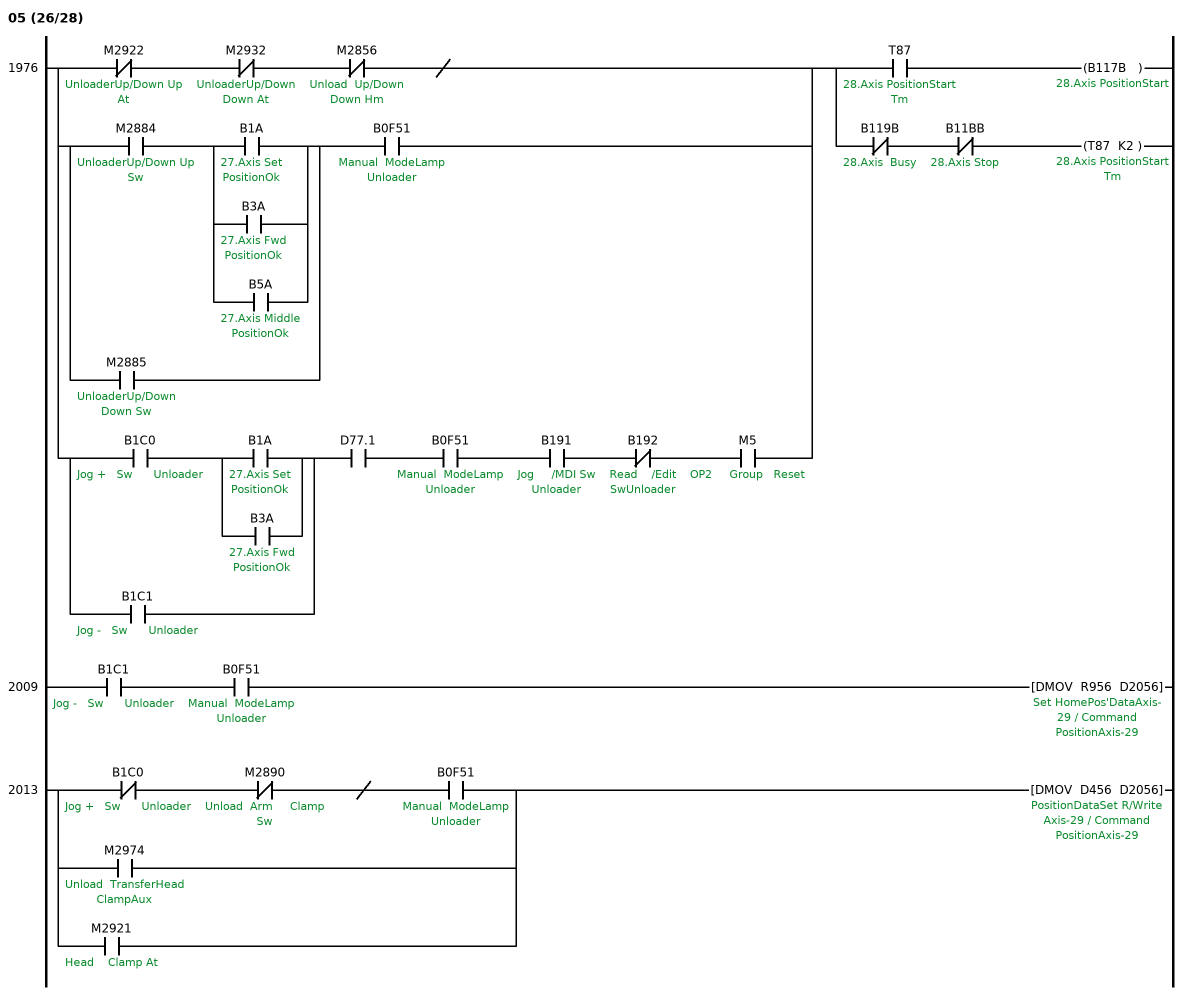
1976  LDI     M2922  ; UnloaderUp/Down Up At
      ANI     M2932  ; UnloaderUp/Down Down At
      ANI     M2856  ; Unload  Up/Down Down Hm
      INV
      LD      M2884  ; UnloaderUp/Down Up Sw
      LD      B1A  ; 27.Axis Set     PositionOk
      OR      B3A  ; 27.Axis Fwd     PositionOk
      OR      B5A  ; 27.Axis Middle  PositionOk
      ANB
      OR      M2885  ; UnloaderUp/Down Down Sw
      AND     B0F51  ; Manual  ModeLampUnloader
      ORB
      LD      B1C0  ; Jog +   Sw      Unloader
      LD      B1A  ; 27.Axis Set     PositionOk
      OR      B3A  ; 27.Axis Fwd     PositionOk
      ANB
      OR      B1C1  ; Jog -   Sw      Unloader
      AND     D77.1
      AND     B0F51  ; Manual  ModeLampUnloader
      AND     B191  ; Jog     /MDI Sw Unloader
      ANI     B192  ; Read    /Edit SwUnloader
      AND     M5  ; OP2     Group   Reset
      ORB
      MPS
      AND     T87  ; 28.Axis PositionStart Tm
      OUT     B117B  ; 28.Axis PositionStart
      MPP
      ANI     B119B  ; 28.Axis  Busy
      ANI     B11BB  ; 28.Axis Stop
      OUT     T87 K2  ; 28.Axis PositionStart Tm
2009  LD      B1C1  ; Jog -   Sw      Unloader
      AND     B0F51  ; Manual  ModeLampUnloader
      DMOV    R956 D2056  ; Set HomePos'DataAxis-29 / Command PositionAxis-29
2013  LDI     B1C0  ; Jog +   Sw      Unloader
      ANI     M2890  ; Unload  Arm     Clamp Sw
      INV
      AND     B0F51  ; Manual  ModeLampUnloader
      OR      M2974  ; Unload  TransferHead    ClampAux
      OR      M2921  ; Head    Clamp At
      DMOV    D456 D2056  ; PositionDataSet R/Write Axis-29
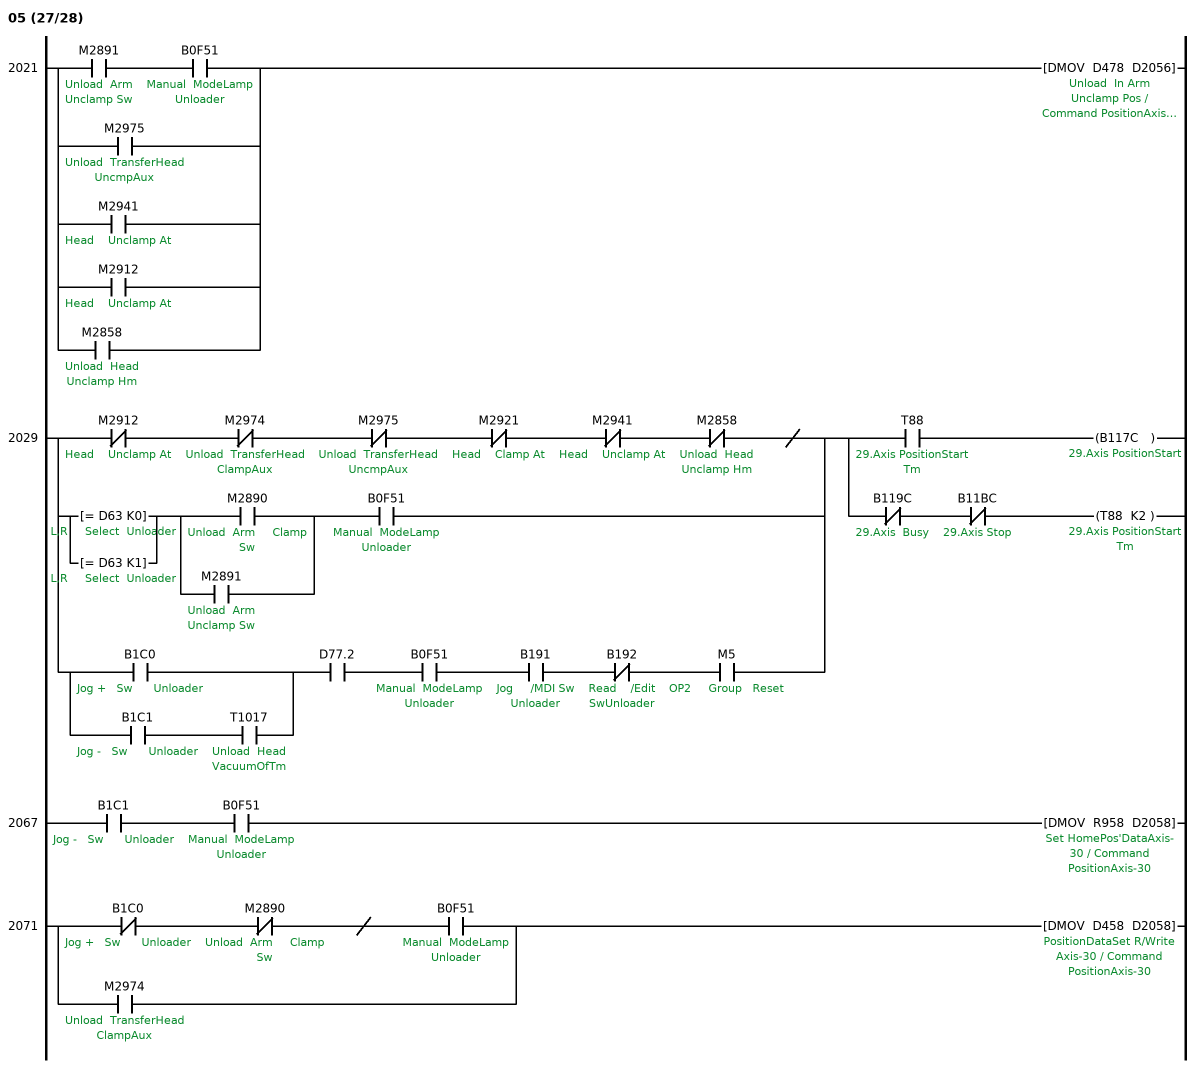
2021  LD      M2891  ; Unload  Arm     Unclamp Sw
      AND     B0F51  ; Manual  ModeLampUnloader
      OR      M2975  ; Unload  TransferHead    UncmpAux
      OR      M2941  ; Head    Unclamp At
      OR      M2912  ; Head    Unclamp At
      OR      M2858  ; Unload  Head    Unclamp Hm
      DMOV    D478 D2056  ; Unload  In Arm  Unclamp Pos
2029  LDI     M2912  ; Head    Unclamp At
      ANI     M2974  ; Unload  TransferHead    ClampAux
      ANI     M2975  ; Unload  TransferHead    UncmpAux
      ANI     M2921  ; Head    Clamp At
      ANI     M2941  ; Head    Unclamp At
      ANI     M2858  ; Unload  Head    Unclamp Hm
      INV
      LD=     D63 K0  ; L,R     Select  Unloader
      OR=     D63 K1  ; L,R     Select  Unloader
      LD      M2890  ; Unload  Arm     Clamp Sw
      OR      M2891  ; Unload  Arm     Unclamp Sw
      ANB
      AND     B0F51  ; Manual  ModeLampUnloader
      ORB
      LD      B1C0  ; Jog +   Sw      Unloader
      LD      B1C1  ; Jog -   Sw      Unloader
      AND     T1017  ; Unload  Head    VacuumOfTm
      ORB
      AND     D77.2
      AND     B0F51  ; Manual  ModeLampUnloader
      AND     B191  ; Jog     /MDI Sw Unloader
      ANI     B192  ; Read    /Edit SwUnloader
      AND     M5  ; OP2     Group   Reset
      ORB
      MPS
      AND     T88  ; 29.Axis PositionStart Tm
      OUT     B117C  ; 29.Axis PositionStart
      MPP
      ANI     B119C  ; 29.Axis  Busy
      ANI     B11BC  ; 29.Axis Stop
      OUT     T88 K2  ; 29.Axis PositionStart Tm
2067  LD      B1C1  ; Jog -   Sw      Unloader
      AND     B0F51  ; Manual  ModeLampUnloader
      DMOV    R958 D2058  ; Set HomePos'DataAxis-30 / Command PositionAxis-30
2071  LDI     B1C0  ; Jog +   Sw      Unloader
      ANI     M2890  ; Unload  Arm     Clamp Sw
      INV
      AND     B0F51  ; Manual  ModeLampUnloader
      OR      M2974  ; Unload  TransferHead    ClampAux
      DMOV    D458 D2058  ; PositionDataSet R/Write Axis-30
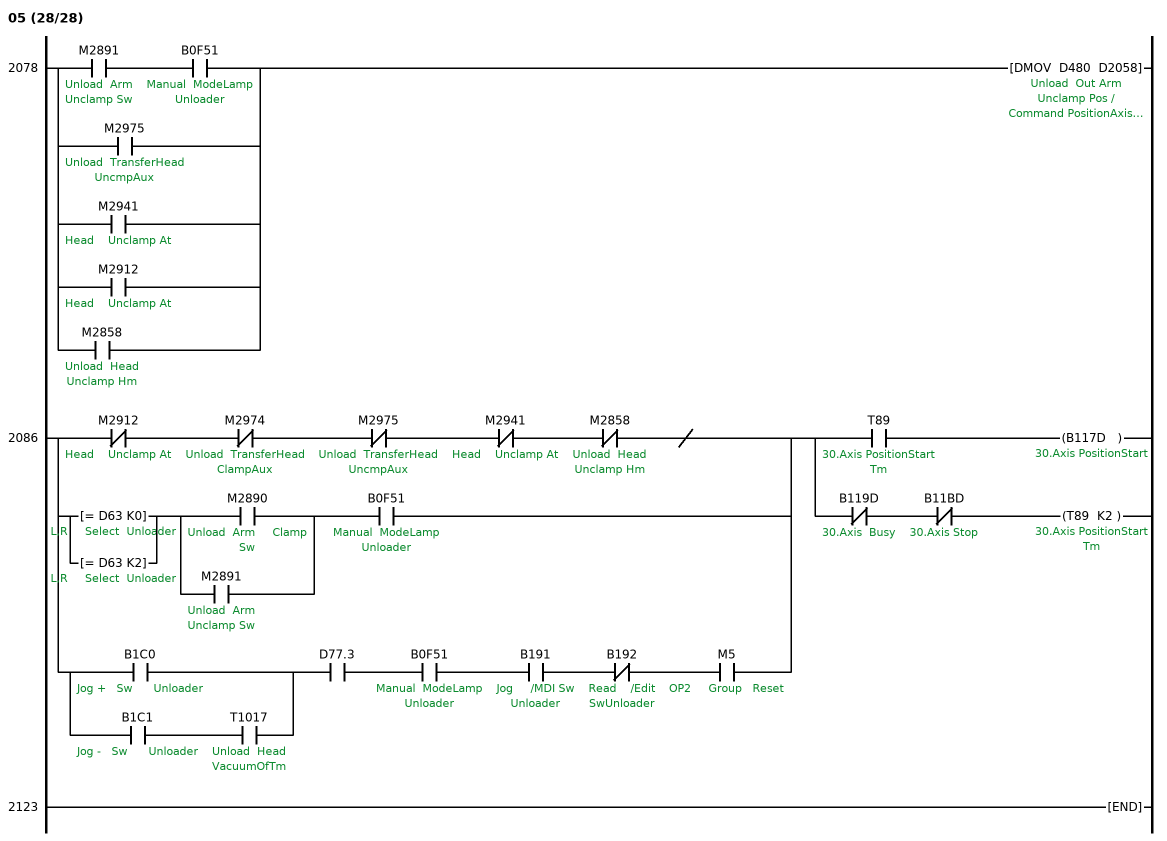
2078  LD      M2891  ; Unload  Arm     Unclamp Sw
      AND     B0F51  ; Manual  ModeLampUnloader
      OR      M2975  ; Unload  TransferHead    UncmpAux
      OR      M2941  ; Head    Unclamp At
      OR      M2912  ; Head    Unclamp At
      OR      M2858  ; Unload  Head    Unclamp Hm
      DMOV    D480 D2058  ; Unload  Out Arm Unclamp Pos
2086  LDI     M2912  ; Head    Unclamp At
      ANI     M2974  ; Unload  TransferHead    ClampAux
      ANI     M2975  ; Unload  TransferHead    UncmpAux
      ANI     M2941  ; Head    Unclamp At
      ANI     M2858  ; Unload  Head    Unclamp Hm
      INV
      LD=     D63 K0  ; L,R     Select  Unloader
      OR=     D63 K2  ; L,R     Select  Unloader
      LD      M2890  ; Unload  Arm     Clamp Sw
      OR      M2891  ; Unload  Arm     Unclamp Sw
      ANB
      AND     B0F51  ; Manual  ModeLampUnloader
      ORB
      LD      B1C0  ; Jog +   Sw      Unloader
      LD      B1C1  ; Jog -   Sw      Unloader
      AND     T1017  ; Unload  Head    VacuumOfTm
      ORB
      AND     D77.3
      AND     B0F51  ; Manual  ModeLampUnloader
      AND     B191  ; Jog     /MDI Sw Unloader
      ANI     B192  ; Read    /Edit SwUnloader
      AND     M5  ; OP2     Group   Reset
      ORB
      MPS
      AND     T89  ; 30.Axis PositionStart Tm
      OUT     B117D  ; 30.Axis PositionStart
      MPP
      ANI     B119D  ; 30.Axis  Busy
      ANI     B11BD  ; 30.Axis Stop
      OUT     T89 K2  ; 30.Axis PositionStart Tm
2123  END
END_PROGRAM

PROGRAM 06  // Servo Part
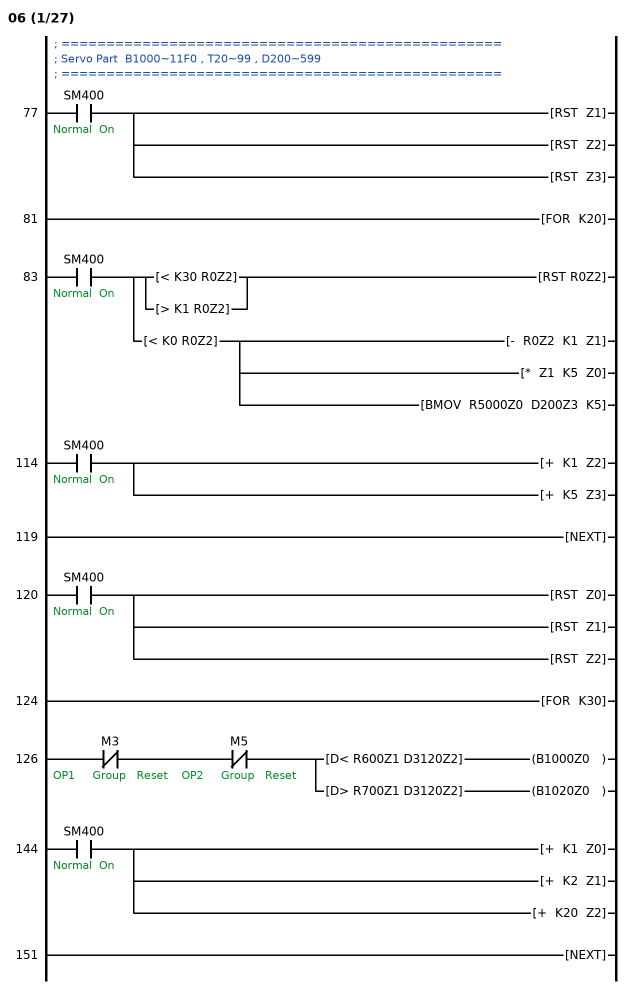
; =================================================
; Servo Part  B1000~11F0 , T20~99 , D200~599
; =================================================
77    LD      SM400  ; Normal  On
      RST     Z1
      RST     Z2
      RST     Z3
81    FOR     K20
83    LD      SM400  ; Normal  On
      MPS
      LD<     K30 R0Z2
      OR>     K1 R0Z2
      ANB
      RST     R0Z2
      MPP
      AND<    K0 R0Z2
      -       R0Z2 K1 Z1
      *       Z1 K5 Z0
      BMOV    R5000Z0 D200Z3 K5
114   LD      SM400  ; Normal  On
      +       K1 Z2
      +       K5 Z3
119   NEXT
120   LD      SM400  ; Normal  On
      RST     Z0
      RST     Z1
      RST     Z2
124   FOR     K30
126   LDI     M3  ; OP1     Group   Reset
      ANI     M5  ; OP2     Group   Reset
      MPS
      ANDD<   R600Z1 D3120Z2
      OUT     B1000Z0
      MPP
      ANDD>   R700Z1 D3120Z2
      OUT     B1020Z0
144   LD      SM400  ; Normal  On
      +       K1 Z0
      +       K2 Z1
      +       K20 Z2
151   NEXT
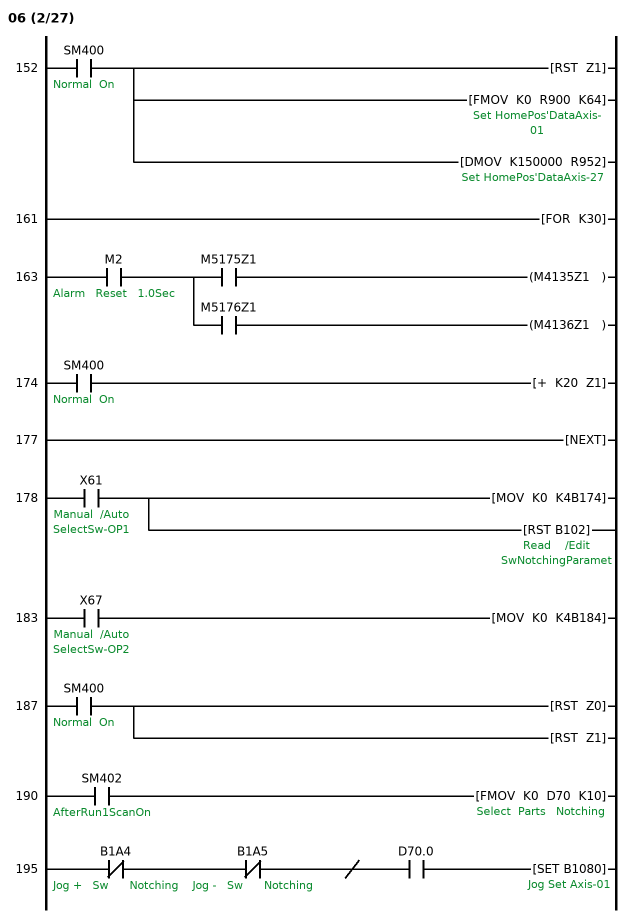
152   LD      SM400  ; Normal  On
      RST     Z1
      FMOV    K0 R900 K64  ; Set HomePos'DataAxis-01
      DMOV    K150000 R952  ; Set HomePos'DataAxis-27
161   FOR     K30
163   LD      M2  ; Alarm   Reset   1.0Sec
      MPS
      AND     M5175Z1
      OUT     M4135Z1
      MPP
      AND     M5176Z1
      OUT     M4136Z1
174   LD      SM400  ; Normal  On
      +       K20 Z1
177   NEXT
178   LD      X61  ; Manual  /Auto   SelectSw-OP1
      MOV     K0 K4B174  ; Jog FastSpeed SwNotching
      RST     B102  ; Read    /Edit SwNotchingParamet
183   LD      X67  ; Manual  /Auto   SelectSw-OP2
      MOV     K0 K4B184  ; Jog FastSpeed SwL & Z
187   LD      SM400  ; Normal  On
      RST     Z0
      RST     Z1
190   LD      SM402  ; AfterRun1ScanOn
      FMOV    K0 D70 K10  ; Select  Parts   Notching
195   LDI     B1A4  ; Jog +   Sw      Notching
      ANI     B1A5  ; Jog -   Sw      Notching
      INV
      AND     D70.0
      SET     B1080  ; Jog Set Axis-01
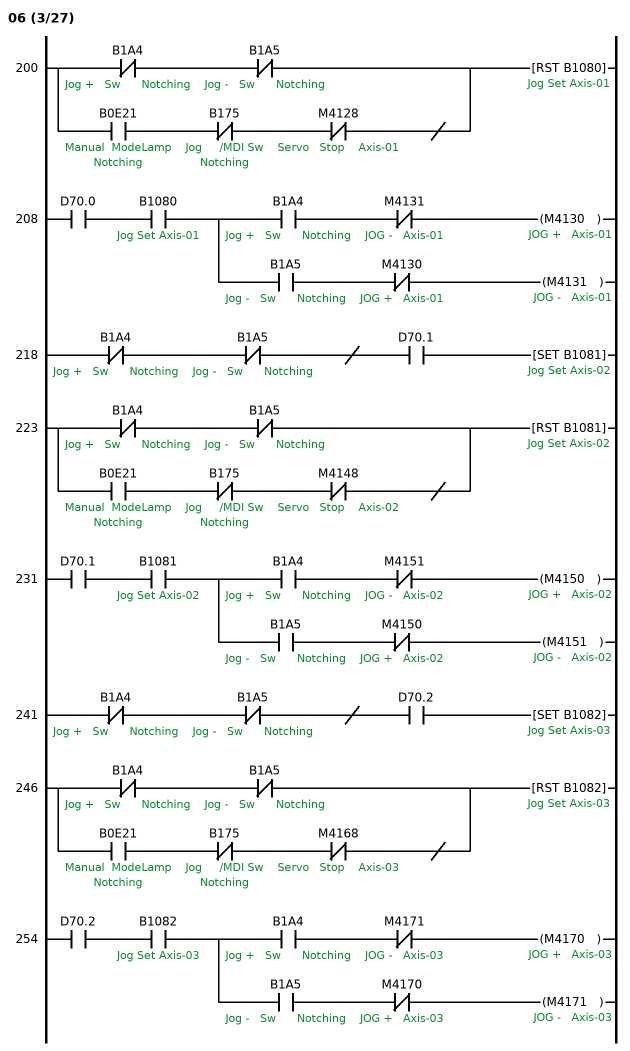
200   LDI     B1A4  ; Jog +   Sw      Notching
      ANI     B1A5  ; Jog -   Sw      Notching
      LD      B0E21  ; Manual  ModeLampNotching
      ANI     B175  ; Jog     /MDI Sw Notching
      ANI     M4128  ; Servo   Stop    Axis-01
      INV
      ORB
      RST     B1080  ; Jog Set Axis-01
208   LD      D70.0
      AND     B1080  ; Jog Set Axis-01
      MPS
      AND     B1A4  ; Jog +   Sw      Notching
      ANI     M4131  ; JOG -   Axis-01
      OUT     M4130  ; JOG +   Axis-01
      MPP
      AND     B1A5  ; Jog -   Sw      Notching
      ANI     M4130  ; JOG +   Axis-01
      OUT     M4131  ; JOG -   Axis-01
218   LDI     B1A4  ; Jog +   Sw      Notching
      ANI     B1A5  ; Jog -   Sw      Notching
      INV
      AND     D70.1
      SET     B1081  ; Jog Set Axis-02
223   LDI     B1A4  ; Jog +   Sw      Notching
      ANI     B1A5  ; Jog -   Sw      Notching
      LD      B0E21  ; Manual  ModeLampNotching
      ANI     B175  ; Jog     /MDI Sw Notching
      ANI     M4148  ; Servo   Stop    Axis-02
      INV
      ORB
      RST     B1081  ; Jog Set Axis-02
231   LD      D70.1
      AND     B1081  ; Jog Set Axis-02
      MPS
      AND     B1A4  ; Jog +   Sw      Notching
      ANI     M4151  ; JOG -   Axis-02
      OUT     M4150  ; JOG +   Axis-02
      MPP
      AND     B1A5  ; Jog -   Sw      Notching
      ANI     M4150  ; JOG +   Axis-02
      OUT     M4151  ; JOG -   Axis-02
241   LDI     B1A4  ; Jog +   Sw      Notching
      ANI     B1A5  ; Jog -   Sw      Notching
      INV
      AND     D70.2
      SET     B1082  ; Jog Set Axis-03
246   LDI     B1A4  ; Jog +   Sw      Notching
      ANI     B1A5  ; Jog -   Sw      Notching
      LD      B0E21  ; Manual  ModeLampNotching
      ANI     B175  ; Jog     /MDI Sw Notching
      ANI     M4168  ; Servo   Stop    Axis-03
      INV
      ORB
      RST     B1082  ; Jog Set Axis-03
254   LD      D70.2
      AND     B1082  ; Jog Set Axis-03
      MPS
      AND     B1A4  ; Jog +   Sw      Notching
      ANI     M4171  ; JOG -   Axis-03
      OUT     M4170  ; JOG +   Axis-03
      MPP
      AND     B1A5  ; Jog -   Sw      Notching
      ANI     M4170  ; JOG +   Axis-03
      OUT     M4171  ; JOG -   Axis-03
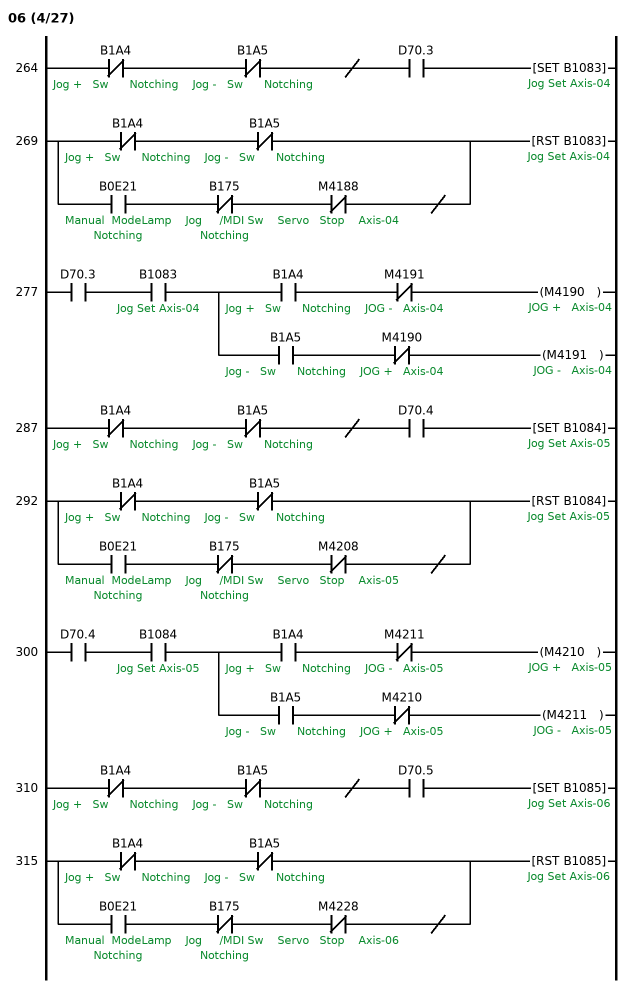
264   LDI     B1A4  ; Jog +   Sw      Notching
      ANI     B1A5  ; Jog -   Sw      Notching
      INV
      AND     D70.3
      SET     B1083  ; Jog Set Axis-04
269   LDI     B1A4  ; Jog +   Sw      Notching
      ANI     B1A5  ; Jog -   Sw      Notching
      LD      B0E21  ; Manual  ModeLampNotching
      ANI     B175  ; Jog     /MDI Sw Notching
      ANI     M4188  ; Servo   Stop    Axis-04
      INV
      ORB
      RST     B1083  ; Jog Set Axis-04
277   LD      D70.3
      AND     B1083  ; Jog Set Axis-04
      MPS
      AND     B1A4  ; Jog +   Sw      Notching
      ANI     M4191  ; JOG -   Axis-04
      OUT     M4190  ; JOG +   Axis-04
      MPP
      AND     B1A5  ; Jog -   Sw      Notching
      ANI     M4190  ; JOG +   Axis-04
      OUT     M4191  ; JOG -   Axis-04
287   LDI     B1A4  ; Jog +   Sw      Notching
      ANI     B1A5  ; Jog -   Sw      Notching
      INV
      AND     D70.4
      SET     B1084  ; Jog Set Axis-05
292   LDI     B1A4  ; Jog +   Sw      Notching
      ANI     B1A5  ; Jog -   Sw      Notching
      LD      B0E21  ; Manual  ModeLampNotching
      ANI     B175  ; Jog     /MDI Sw Notching
      ANI     M4208  ; Servo   Stop    Axis-05
      INV
      ORB
      RST     B1084  ; Jog Set Axis-05
300   LD      D70.4
      AND     B1084  ; Jog Set Axis-05
      MPS
      AND     B1A4  ; Jog +   Sw      Notching
      ANI     M4211  ; JOG -   Axis-05
      OUT     M4210  ; JOG +   Axis-05
      MPP
      AND     B1A5  ; Jog -   Sw      Notching
      ANI     M4210  ; JOG +   Axis-05
      OUT     M4211  ; JOG -   Axis-05
310   LDI     B1A4  ; Jog +   Sw      Notching
      ANI     B1A5  ; Jog -   Sw      Notching
      INV
      AND     D70.5
      SET     B1085  ; Jog Set Axis-06
315   LDI     B1A4  ; Jog +   Sw      Notching
      ANI     B1A5  ; Jog -   Sw      Notching
      LD      B0E21  ; Manual  ModeLampNotching
      ANI     B175  ; Jog     /MDI Sw Notching
      ANI     M4228  ; Servo   Stop    Axis-06
      INV
      ORB
      RST     B1085  ; Jog Set Axis-06
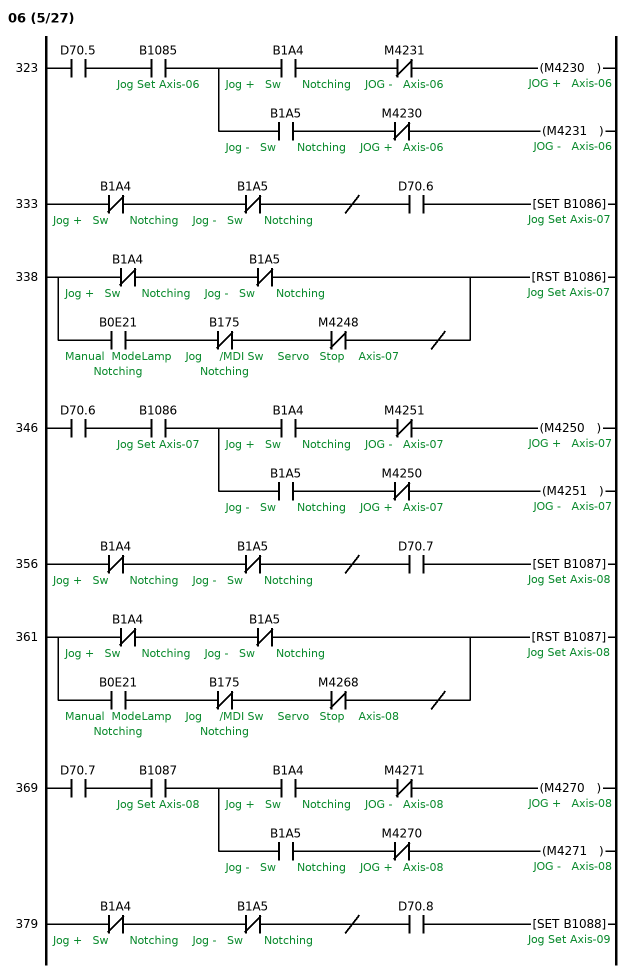
323   LD      D70.5
      AND     B1085  ; Jog Set Axis-06
      MPS
      AND     B1A4  ; Jog +   Sw      Notching
      ANI     M4231  ; JOG -   Axis-06
      OUT     M4230  ; JOG +   Axis-06
      MPP
      AND     B1A5  ; Jog -   Sw      Notching
      ANI     M4230  ; JOG +   Axis-06
      OUT     M4231  ; JOG -   Axis-06
333   LDI     B1A4  ; Jog +   Sw      Notching
      ANI     B1A5  ; Jog -   Sw      Notching
      INV
      AND     D70.6
      SET     B1086  ; Jog Set Axis-07
338   LDI     B1A4  ; Jog +   Sw      Notching
      ANI     B1A5  ; Jog -   Sw      Notching
      LD      B0E21  ; Manual  ModeLampNotching
      ANI     B175  ; Jog     /MDI Sw Notching
      ANI     M4248  ; Servo   Stop    Axis-07
      INV
      ORB
      RST     B1086  ; Jog Set Axis-07
346   LD      D70.6
      AND     B1086  ; Jog Set Axis-07
      MPS
      AND     B1A4  ; Jog +   Sw      Notching
      ANI     M4251  ; JOG -   Axis-07
      OUT     M4250  ; JOG +   Axis-07
      MPP
      AND     B1A5  ; Jog -   Sw      Notching
      ANI     M4250  ; JOG +   Axis-07
      OUT     M4251  ; JOG -   Axis-07
356   LDI     B1A4  ; Jog +   Sw      Notching
      ANI     B1A5  ; Jog -   Sw      Notching
      INV
      AND     D70.7
      SET     B1087  ; Jog Set Axis-08
361   LDI     B1A4  ; Jog +   Sw      Notching
      ANI     B1A5  ; Jog -   Sw      Notching
      LD      B0E21  ; Manual  ModeLampNotching
      ANI     B175  ; Jog     /MDI Sw Notching
      ANI     M4268  ; Servo   Stop    Axis-08
      INV
      ORB
      RST     B1087  ; Jog Set Axis-08
369   LD      D70.7
      AND     B1087  ; Jog Set Axis-08
      MPS
      AND     B1A4  ; Jog +   Sw      Notching
      ANI     M4271  ; JOG -   Axis-08
      OUT     M4270  ; JOG +   Axis-08
      MPP
      AND     B1A5  ; Jog -   Sw      Notching
      ANI     M4270  ; JOG +   Axis-08
      OUT     M4271  ; JOG -   Axis-08
379   LDI     B1A4  ; Jog +   Sw      Notching
      ANI     B1A5  ; Jog -   Sw      Notching
      INV
      AND     D70.8
      SET     B1088  ; Jog Set Axis-09
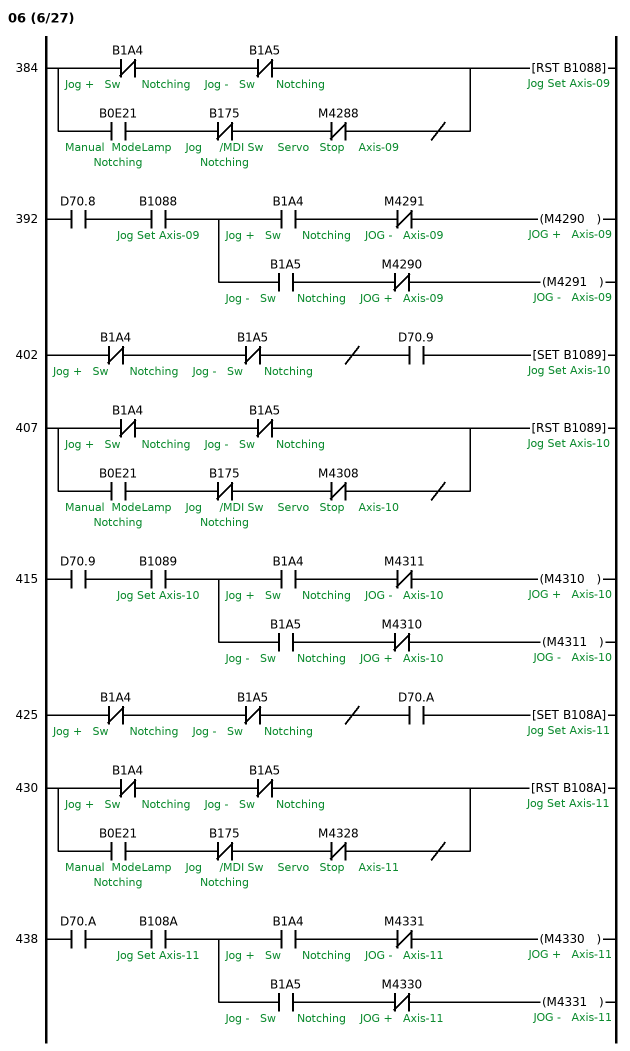
384   LDI     B1A4  ; Jog +   Sw      Notching
      ANI     B1A5  ; Jog -   Sw      Notching
      LD      B0E21  ; Manual  ModeLampNotching
      ANI     B175  ; Jog     /MDI Sw Notching
      ANI     M4288  ; Servo   Stop    Axis-09
      INV
      ORB
      RST     B1088  ; Jog Set Axis-09
392   LD      D70.8
      AND     B1088  ; Jog Set Axis-09
      MPS
      AND     B1A4  ; Jog +   Sw      Notching
      ANI     M4291  ; JOG -   Axis-09
      OUT     M4290  ; JOG +   Axis-09
      MPP
      AND     B1A5  ; Jog -   Sw      Notching
      ANI     M4290  ; JOG +   Axis-09
      OUT     M4291  ; JOG -   Axis-09
402   LDI     B1A4  ; Jog +   Sw      Notching
      ANI     B1A5  ; Jog -   Sw      Notching
      INV
      AND     D70.9
      SET     B1089  ; Jog Set Axis-10
407   LDI     B1A4  ; Jog +   Sw      Notching
      ANI     B1A5  ; Jog -   Sw      Notching
      LD      B0E21  ; Manual  ModeLampNotching
      ANI     B175  ; Jog     /MDI Sw Notching
      ANI     M4308  ; Servo   Stop    Axis-10
      INV
      ORB
      RST     B1089  ; Jog Set Axis-10
415   LD      D70.9
      AND     B1089  ; Jog Set Axis-10
      MPS
      AND     B1A4  ; Jog +   Sw      Notching
      ANI     M4311  ; JOG -   Axis-10
      OUT     M4310  ; JOG +   Axis-10
      MPP
      AND     B1A5  ; Jog -   Sw      Notching
      ANI     M4310  ; JOG +   Axis-10
      OUT     M4311  ; JOG -   Axis-10
425   LDI     B1A4  ; Jog +   Sw      Notching
      ANI     B1A5  ; Jog -   Sw      Notching
      INV
      AND     D70.A
      SET     B108A  ; Jog Set Axis-11
430   LDI     B1A4  ; Jog +   Sw      Notching
      ANI     B1A5  ; Jog -   Sw      Notching
      LD      B0E21  ; Manual  ModeLampNotching
      ANI     B175  ; Jog     /MDI Sw Notching
      ANI     M4328  ; Servo   Stop    Axis-11
      INV
      ORB
      RST     B108A  ; Jog Set Axis-11
438   LD      D70.A
      AND     B108A  ; Jog Set Axis-11
      MPS
      AND     B1A4  ; Jog +   Sw      Notching
      ANI     M4331  ; JOG -   Axis-11
      OUT     M4330  ; JOG +   Axis-11
      MPP
      AND     B1A5  ; Jog -   Sw      Notching
      ANI     M4330  ; JOG +   Axis-11
      OUT     M4331  ; JOG -   Axis-11
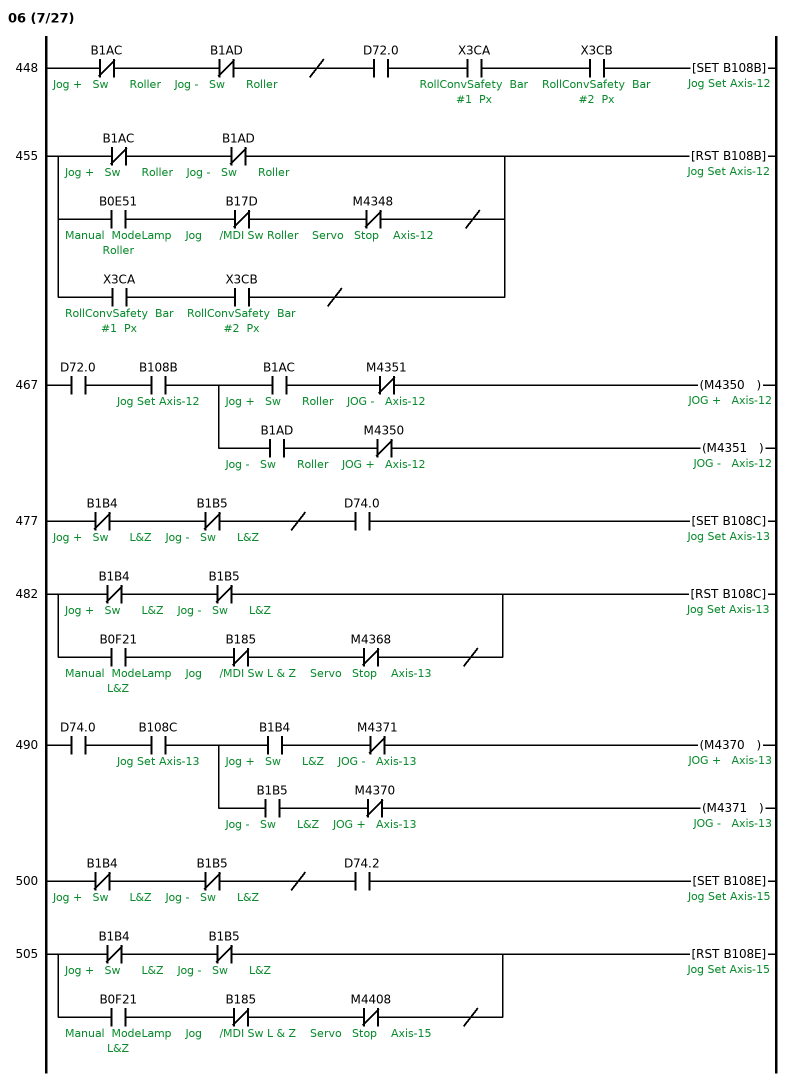
448   LDI     B1AC  ; Jog +   Sw      Roller
      ANI     B1AD  ; Jog -   Sw      Roller
      INV
      AND     D72.0
      AND     X3CA  ; RollConvSafety  Bar #1  Px
      AND     X3CB  ; RollConvSafety  Bar #2  Px
      SET     B108B  ; Jog Set Axis-12
455   LDI     B1AC  ; Jog +   Sw      Roller
      ANI     B1AD  ; Jog -   Sw      Roller
      LD      B0E51  ; Manual  ModeLampRoller
      ANI     B17D  ; Jog     /MDI Sw Roller
      ANI     M4348  ; Servo   Stop    Axis-12
      INV
      ORB
      LD      X3CA  ; RollConvSafety  Bar #1  Px
      AND     X3CB  ; RollConvSafety  Bar #2  Px
      INV
      ORB
      RST     B108B  ; Jog Set Axis-12
467   LD      D72.0
      AND     B108B  ; Jog Set Axis-12
      MPS
      AND     B1AC  ; Jog +   Sw      Roller
      ANI     M4351  ; JOG -   Axis-12
      OUT     M4350  ; JOG +   Axis-12
      MPP
      AND     B1AD  ; Jog -   Sw      Roller
      ANI     M4350  ; JOG +   Axis-12
      OUT     M4351  ; JOG -   Axis-12
477   LDI     B1B4  ; Jog +   Sw      L&Z
      ANI     B1B5  ; Jog -   Sw      L&Z
      INV
      AND     D74.0
      SET     B108C  ; Jog Set Axis-13
482   LDI     B1B4  ; Jog +   Sw      L&Z
      ANI     B1B5  ; Jog -   Sw      L&Z
      LD      B0F21  ; Manual  ModeLampL&Z
      ANI     B185  ; Jog     /MDI Sw L & Z
      ANI     M4368  ; Servo   Stop    Axis-13
      INV
      ORB
      RST     B108C  ; Jog Set Axis-13
490   LD      D74.0
      AND     B108C  ; Jog Set Axis-13
      MPS
      AND     B1B4  ; Jog +   Sw      L&Z
      ANI     M4371  ; JOG -   Axis-13
      OUT     M4370  ; JOG +   Axis-13
      MPP
      AND     B1B5  ; Jog -   Sw      L&Z
      ANI     M4370  ; JOG +   Axis-13
      OUT     M4371  ; JOG -   Axis-13
500   LDI     B1B4  ; Jog +   Sw      L&Z
      ANI     B1B5  ; Jog -   Sw      L&Z
      INV
      AND     D74.2
      SET     B108E  ; Jog Set Axis-15
505   LDI     B1B4  ; Jog +   Sw      L&Z
      ANI     B1B5  ; Jog -   Sw      L&Z
      LD      B0F21  ; Manual  ModeLampL&Z
      ANI     B185  ; Jog     /MDI Sw L & Z
      ANI     M4408  ; Servo   Stop    Axis-15
      INV
      ORB
      RST     B108E  ; Jog Set Axis-15
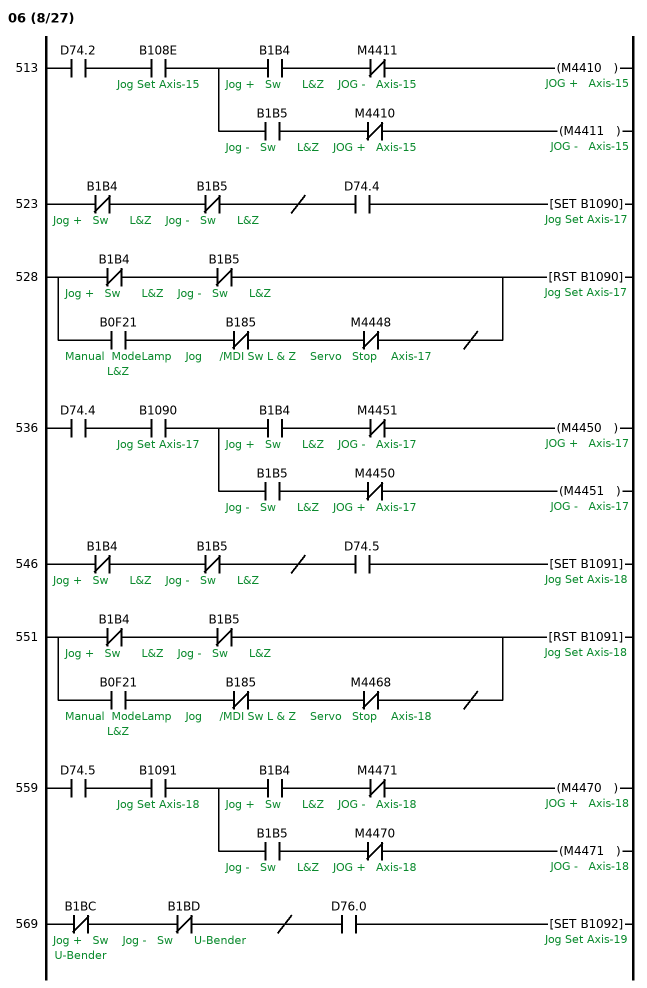
513   LD      D74.2
      AND     B108E  ; Jog Set Axis-15
      MPS
      AND     B1B4  ; Jog +   Sw      L&Z
      ANI     M4411  ; JOG -   Axis-15
      OUT     M4410  ; JOG +   Axis-15
      MPP
      AND     B1B5  ; Jog -   Sw      L&Z
      ANI     M4410  ; JOG +   Axis-15
      OUT     M4411  ; JOG -   Axis-15
523   LDI     B1B4  ; Jog +   Sw      L&Z
      ANI     B1B5  ; Jog -   Sw      L&Z
      INV
      AND     D74.4
      SET     B1090  ; Jog Set Axis-17
528   LDI     B1B4  ; Jog +   Sw      L&Z
      ANI     B1B5  ; Jog -   Sw      L&Z
      LD      B0F21  ; Manual  ModeLampL&Z
      ANI     B185  ; Jog     /MDI Sw L & Z
      ANI     M4448  ; Servo   Stop    Axis-17
      INV
      ORB
      RST     B1090  ; Jog Set Axis-17
536   LD      D74.4
      AND     B1090  ; Jog Set Axis-17
      MPS
      AND     B1B4  ; Jog +   Sw      L&Z
      ANI     M4451  ; JOG -   Axis-17
      OUT     M4450  ; JOG +   Axis-17
      MPP
      AND     B1B5  ; Jog -   Sw      L&Z
      ANI     M4450  ; JOG +   Axis-17
      OUT     M4451  ; JOG -   Axis-17
546   LDI     B1B4  ; Jog +   Sw      L&Z
      ANI     B1B5  ; Jog -   Sw      L&Z
      INV
      AND     D74.5
      SET     B1091  ; Jog Set Axis-18
551   LDI     B1B4  ; Jog +   Sw      L&Z
      ANI     B1B5  ; Jog -   Sw      L&Z
      LD      B0F21  ; Manual  ModeLampL&Z
      ANI     B185  ; Jog     /MDI Sw L & Z
      ANI     M4468  ; Servo   Stop    Axis-18
      INV
      ORB
      RST     B1091  ; Jog Set Axis-18
559   LD      D74.5
      AND     B1091  ; Jog Set Axis-18
      MPS
      AND     B1B4  ; Jog +   Sw      L&Z
      ANI     M4471  ; JOG -   Axis-18
      OUT     M4470  ; JOG +   Axis-18
      MPP
      AND     B1B5  ; Jog -   Sw      L&Z
      ANI     M4470  ; JOG +   Axis-18
      OUT     M4471  ; JOG -   Axis-18
569   LDI     B1BC  ; Jog +   Sw      U-Bender
      ANI     B1BD  ; Jog -   Sw      U-Bender
      INV
      AND     D76.0
      SET     B1092  ; Jog Set Axis-19
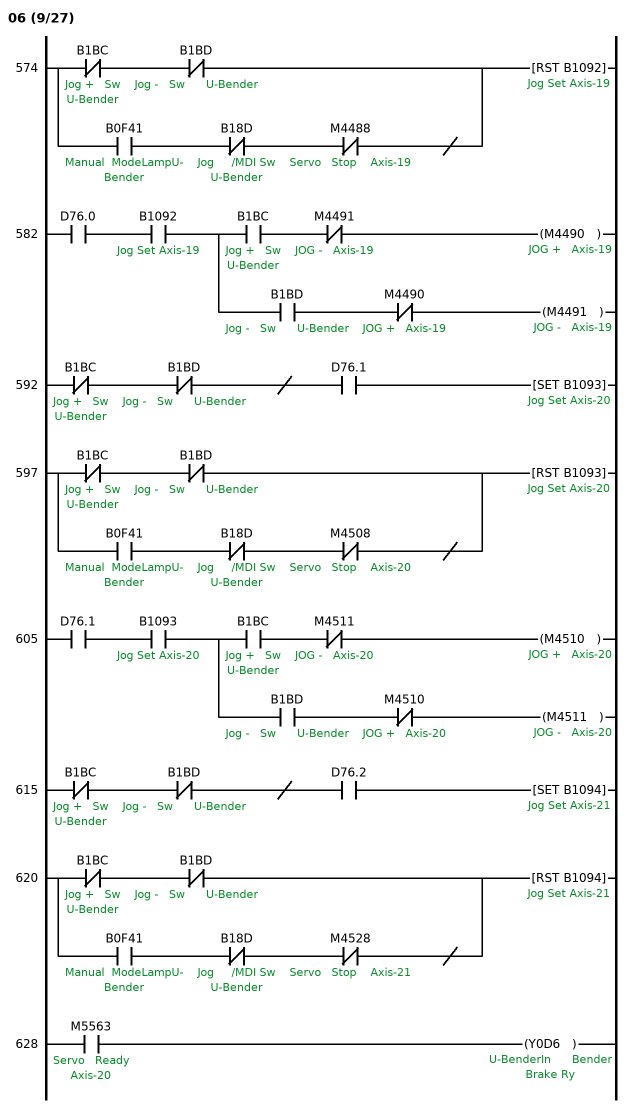
574   LDI     B1BC  ; Jog +   Sw      U-Bender
      ANI     B1BD  ; Jog -   Sw      U-Bender
      LD      B0F41  ; Manual  ModeLampU-Bender
      ANI     B18D  ; Jog     /MDI Sw U-Bender
      ANI     M4488  ; Servo   Stop    Axis-19
      INV
      ORB
      RST     B1092  ; Jog Set Axis-19
582   LD      D76.0
      AND     B1092  ; Jog Set Axis-19
      MPS
      AND     B1BC  ; Jog +   Sw      U-Bender
      ANI     M4491  ; JOG -   Axis-19
      OUT     M4490  ; JOG +   Axis-19
      MPP
      AND     B1BD  ; Jog -   Sw      U-Bender
      ANI     M4490  ; JOG +   Axis-19
      OUT     M4491  ; JOG -   Axis-19
592   LDI     B1BC  ; Jog +   Sw      U-Bender
      ANI     B1BD  ; Jog -   Sw      U-Bender
      INV
      AND     D76.1
      SET     B1093  ; Jog Set Axis-20
597   LDI     B1BC  ; Jog +   Sw      U-Bender
      ANI     B1BD  ; Jog -   Sw      U-Bender
      LD      B0F41  ; Manual  ModeLampU-Bender
      ANI     B18D  ; Jog     /MDI Sw U-Bender
      ANI     M4508  ; Servo   Stop    Axis-20
      INV
      ORB
      RST     B1093  ; Jog Set Axis-20
605   LD      D76.1
      AND     B1093  ; Jog Set Axis-20
      MPS
      AND     B1BC  ; Jog +   Sw      U-Bender
      ANI     M4511  ; JOG -   Axis-20
      OUT     M4510  ; JOG +   Axis-20
      MPP
      AND     B1BD  ; Jog -   Sw      U-Bender
      ANI     M4510  ; JOG +   Axis-20
      OUT     M4511  ; JOG -   Axis-20
615   LDI     B1BC  ; Jog +   Sw      U-Bender
      ANI     B1BD  ; Jog -   Sw      U-Bender
      INV
      AND     D76.2
      SET     B1094  ; Jog Set Axis-21
620   LDI     B1BC  ; Jog +   Sw      U-Bender
      ANI     B1BD  ; Jog -   Sw      U-Bender
      LD      B0F41  ; Manual  ModeLampU-Bender
      ANI     B18D  ; Jog     /MDI Sw U-Bender
      ANI     M4528  ; Servo   Stop    Axis-21
      INV
      ORB
      RST     B1094  ; Jog Set Axis-21
628   LD      M5563  ; Servo   Ready   Axis-20
      OUT     Y0D6  ; U-BenderIn      Bender  Brake Ry
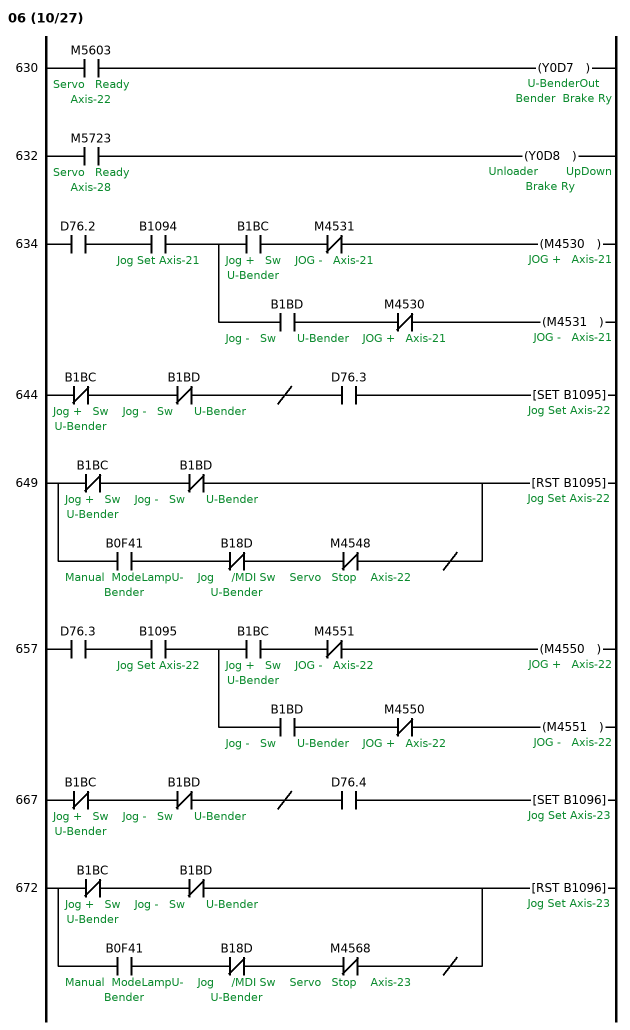
630   LD      M5603  ; Servo   Ready   Axis-22
      OUT     Y0D7  ; U-BenderOut     Bender  Brake Ry
632   LD      M5723  ; Servo   Ready   Axis-28
      OUT     Y0D8  ; Unloader        UpDown  Brake Ry
634   LD      D76.2
      AND     B1094  ; Jog Set Axis-21
      MPS
      AND     B1BC  ; Jog +   Sw      U-Bender
      ANI     M4531  ; JOG -   Axis-21
      OUT     M4530  ; JOG +   Axis-21
      MPP
      AND     B1BD  ; Jog -   Sw      U-Bender
      ANI     M4530  ; JOG +   Axis-21
      OUT     M4531  ; JOG -   Axis-21
644   LDI     B1BC  ; Jog +   Sw      U-Bender
      ANI     B1BD  ; Jog -   Sw      U-Bender
      INV
      AND     D76.3
      SET     B1095  ; Jog Set Axis-22
649   LDI     B1BC  ; Jog +   Sw      U-Bender
      ANI     B1BD  ; Jog -   Sw      U-Bender
      LD      B0F41  ; Manual  ModeLampU-Bender
      ANI     B18D  ; Jog     /MDI Sw U-Bender
      ANI     M4548  ; Servo   Stop    Axis-22
      INV
      ORB
      RST     B1095  ; Jog Set Axis-22
657   LD      D76.3
      AND     B1095  ; Jog Set Axis-22
      MPS
      AND     B1BC  ; Jog +   Sw      U-Bender
      ANI     M4551  ; JOG -   Axis-22
      OUT     M4550  ; JOG +   Axis-22
      MPP
      AND     B1BD  ; Jog -   Sw      U-Bender
      ANI     M4550  ; JOG +   Axis-22
      OUT     M4551  ; JOG -   Axis-22
667   LDI     B1BC  ; Jog +   Sw      U-Bender
      ANI     B1BD  ; Jog -   Sw      U-Bender
      INV
      AND     D76.4
      SET     B1096  ; Jog Set Axis-23
672   LDI     B1BC  ; Jog +   Sw      U-Bender
      ANI     B1BD  ; Jog -   Sw      U-Bender
      LD      B0F41  ; Manual  ModeLampU-Bender
      ANI     B18D  ; Jog     /MDI Sw U-Bender
      ANI     M4568  ; Servo   Stop    Axis-23
      INV
      ORB
      RST     B1096  ; Jog Set Axis-23
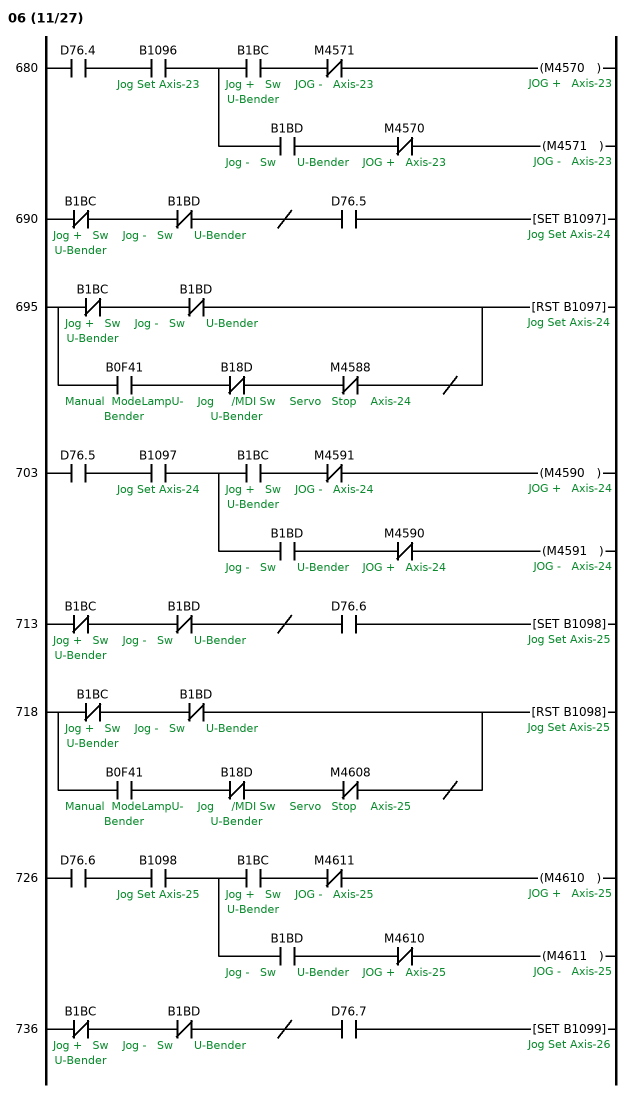
680   LD      D76.4
      AND     B1096  ; Jog Set Axis-23
      MPS
      AND     B1BC  ; Jog +   Sw      U-Bender
      ANI     M4571  ; JOG -   Axis-23
      OUT     M4570  ; JOG +   Axis-23
      MPP
      AND     B1BD  ; Jog -   Sw      U-Bender
      ANI     M4570  ; JOG +   Axis-23
      OUT     M4571  ; JOG -   Axis-23
690   LDI     B1BC  ; Jog +   Sw      U-Bender
      ANI     B1BD  ; Jog -   Sw      U-Bender
      INV
      AND     D76.5
      SET     B1097  ; Jog Set Axis-24
695   LDI     B1BC  ; Jog +   Sw      U-Bender
      ANI     B1BD  ; Jog -   Sw      U-Bender
      LD      B0F41  ; Manual  ModeLampU-Bender
      ANI     B18D  ; Jog     /MDI Sw U-Bender
      ANI     M4588  ; Servo   Stop    Axis-24
      INV
      ORB
      RST     B1097  ; Jog Set Axis-24
703   LD      D76.5
      AND     B1097  ; Jog Set Axis-24
      MPS
      AND     B1BC  ; Jog +   Sw      U-Bender
      ANI     M4591  ; JOG -   Axis-24
      OUT     M4590  ; JOG +   Axis-24
      MPP
      AND     B1BD  ; Jog -   Sw      U-Bender
      ANI     M4590  ; JOG +   Axis-24
      OUT     M4591  ; JOG -   Axis-24
713   LDI     B1BC  ; Jog +   Sw      U-Bender
      ANI     B1BD  ; Jog -   Sw      U-Bender
      INV
      AND     D76.6
      SET     B1098  ; Jog Set Axis-25
718   LDI     B1BC  ; Jog +   Sw      U-Bender
      ANI     B1BD  ; Jog -   Sw      U-Bender
      LD      B0F41  ; Manual  ModeLampU-Bender
      ANI     B18D  ; Jog     /MDI Sw U-Bender
      ANI     M4608  ; Servo   Stop    Axis-25
      INV
      ORB
      RST     B1098  ; Jog Set Axis-25
726   LD      D76.6
      AND     B1098  ; Jog Set Axis-25
      MPS
      AND     B1BC  ; Jog +   Sw      U-Bender
      ANI     M4611  ; JOG -   Axis-25
      OUT     M4610  ; JOG +   Axis-25
      MPP
      AND     B1BD  ; Jog -   Sw      U-Bender
      ANI     M4610  ; JOG +   Axis-25
      OUT     M4611  ; JOG -   Axis-25
736   LDI     B1BC  ; Jog +   Sw      U-Bender
      ANI     B1BD  ; Jog -   Sw      U-Bender
      INV
      AND     D76.7
      SET     B1099  ; Jog Set Axis-26
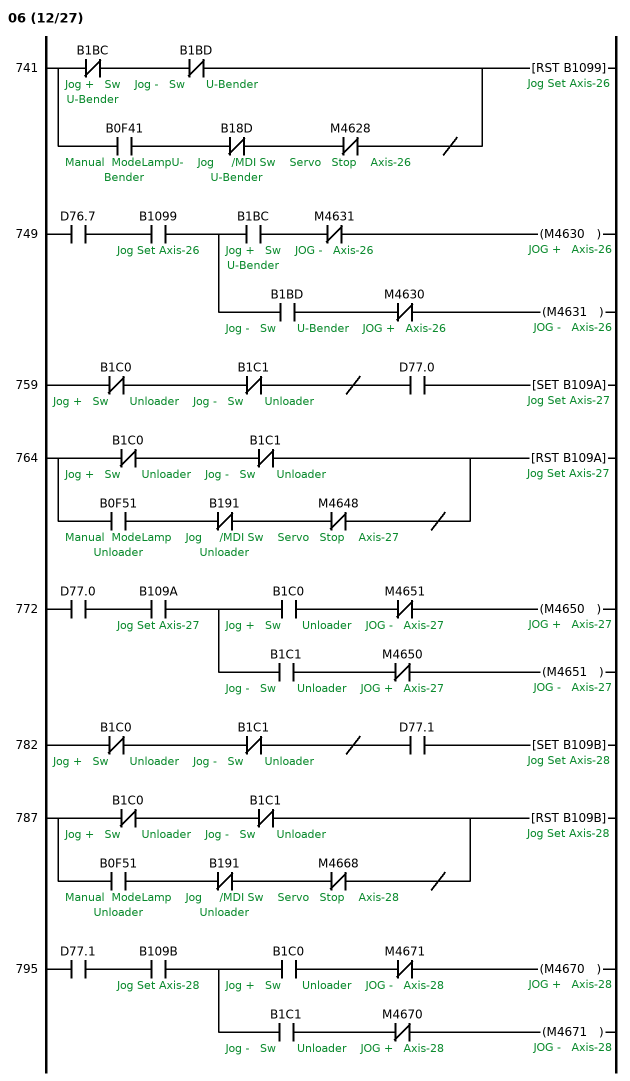
741   LDI     B1BC  ; Jog +   Sw      U-Bender
      ANI     B1BD  ; Jog -   Sw      U-Bender
      LD      B0F41  ; Manual  ModeLampU-Bender
      ANI     B18D  ; Jog     /MDI Sw U-Bender
      ANI     M4628  ; Servo   Stop    Axis-26
      INV
      ORB
      RST     B1099  ; Jog Set Axis-26
749   LD      D76.7
      AND     B1099  ; Jog Set Axis-26
      MPS
      AND     B1BC  ; Jog +   Sw      U-Bender
      ANI     M4631  ; JOG -   Axis-26
      OUT     M4630  ; JOG +   Axis-26
      MPP
      AND     B1BD  ; Jog -   Sw      U-Bender
      ANI     M4630  ; JOG +   Axis-26
      OUT     M4631  ; JOG -   Axis-26
759   LDI     B1C0  ; Jog +   Sw      Unloader
      ANI     B1C1  ; Jog -   Sw      Unloader
      INV
      AND     D77.0
      SET     B109A  ; Jog Set Axis-27
764   LDI     B1C0  ; Jog +   Sw      Unloader
      ANI     B1C1  ; Jog -   Sw      Unloader
      LD      B0F51  ; Manual  ModeLampUnloader
      ANI     B191  ; Jog     /MDI Sw Unloader
      ANI     M4648  ; Servo   Stop    Axis-27
      INV
      ORB
      RST     B109A  ; Jog Set Axis-27
772   LD      D77.0
      AND     B109A  ; Jog Set Axis-27
      MPS
      AND     B1C0  ; Jog +   Sw      Unloader
      ANI     M4651  ; JOG -   Axis-27
      OUT     M4650  ; JOG +   Axis-27
      MPP
      AND     B1C1  ; Jog -   Sw      Unloader
      ANI     M4650  ; JOG +   Axis-27
      OUT     M4651  ; JOG -   Axis-27
782   LDI     B1C0  ; Jog +   Sw      Unloader
      ANI     B1C1  ; Jog -   Sw      Unloader
      INV
      AND     D77.1
      SET     B109B  ; Jog Set Axis-28
787   LDI     B1C0  ; Jog +   Sw      Unloader
      ANI     B1C1  ; Jog -   Sw      Unloader
      LD      B0F51  ; Manual  ModeLampUnloader
      ANI     B191  ; Jog     /MDI Sw Unloader
      ANI     M4668  ; Servo   Stop    Axis-28
      INV
      ORB
      RST     B109B  ; Jog Set Axis-28
795   LD      D77.1
      AND     B109B  ; Jog Set Axis-28
      MPS
      AND     B1C0  ; Jog +   Sw      Unloader
      ANI     M4671  ; JOG -   Axis-28
      OUT     M4670  ; JOG +   Axis-28
      MPP
      AND     B1C1  ; Jog -   Sw      Unloader
      ANI     M4670  ; JOG +   Axis-28
      OUT     M4671  ; JOG -   Axis-28
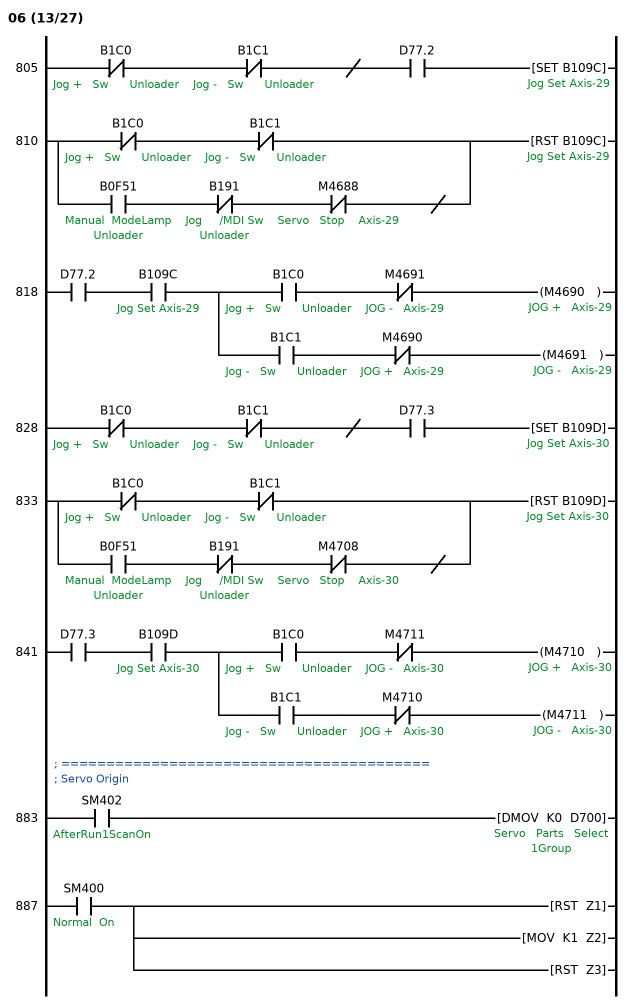
805   LDI     B1C0  ; Jog +   Sw      Unloader
      ANI     B1C1  ; Jog -   Sw      Unloader
      INV
      AND     D77.2
      SET     B109C  ; Jog Set Axis-29
810   LDI     B1C0  ; Jog +   Sw      Unloader
      ANI     B1C1  ; Jog -   Sw      Unloader
      LD      B0F51  ; Manual  ModeLampUnloader
      ANI     B191  ; Jog     /MDI Sw Unloader
      ANI     M4688  ; Servo   Stop    Axis-29
      INV
      ORB
      RST     B109C  ; Jog Set Axis-29
818   LD      D77.2
      AND     B109C  ; Jog Set Axis-29
      MPS
      AND     B1C0  ; Jog +   Sw      Unloader
      ANI     M4691  ; JOG -   Axis-29
      OUT     M4690  ; JOG +   Axis-29
      MPP
      AND     B1C1  ; Jog -   Sw      Unloader
      ANI     M4690  ; JOG +   Axis-29
      OUT     M4691  ; JOG -   Axis-29
828   LDI     B1C0  ; Jog +   Sw      Unloader
      ANI     B1C1  ; Jog -   Sw      Unloader
      INV
      AND     D77.3
      SET     B109D  ; Jog Set Axis-30
833   LDI     B1C0  ; Jog +   Sw      Unloader
      ANI     B1C1  ; Jog -   Sw      Unloader
      LD      B0F51  ; Manual  ModeLampUnloader
      ANI     B191  ; Jog     /MDI Sw Unloader
      ANI     M4708  ; Servo   Stop    Axis-30
      INV
      ORB
      RST     B109D  ; Jog Set Axis-30
841   LD      D77.3
      AND     B109D  ; Jog Set Axis-30
      MPS
      AND     B1C0  ; Jog +   Sw      Unloader
      ANI     M4711  ; JOG -   Axis-30
      OUT     M4710  ; JOG +   Axis-30
      MPP
      AND     B1C1  ; Jog -   Sw      Unloader
      ANI     M4710  ; JOG +   Axis-30
      OUT     M4711  ; JOG -   Axis-30
; =========================================
; Servo Origin
883   LD      SM402  ; AfterRun1ScanOn
      DMOV    K0 D700  ; Servo   Parts   Select  1Group
887   LD      SM400  ; Normal  On
      RST     Z1
      MOV     K1 Z2
      RST     Z3
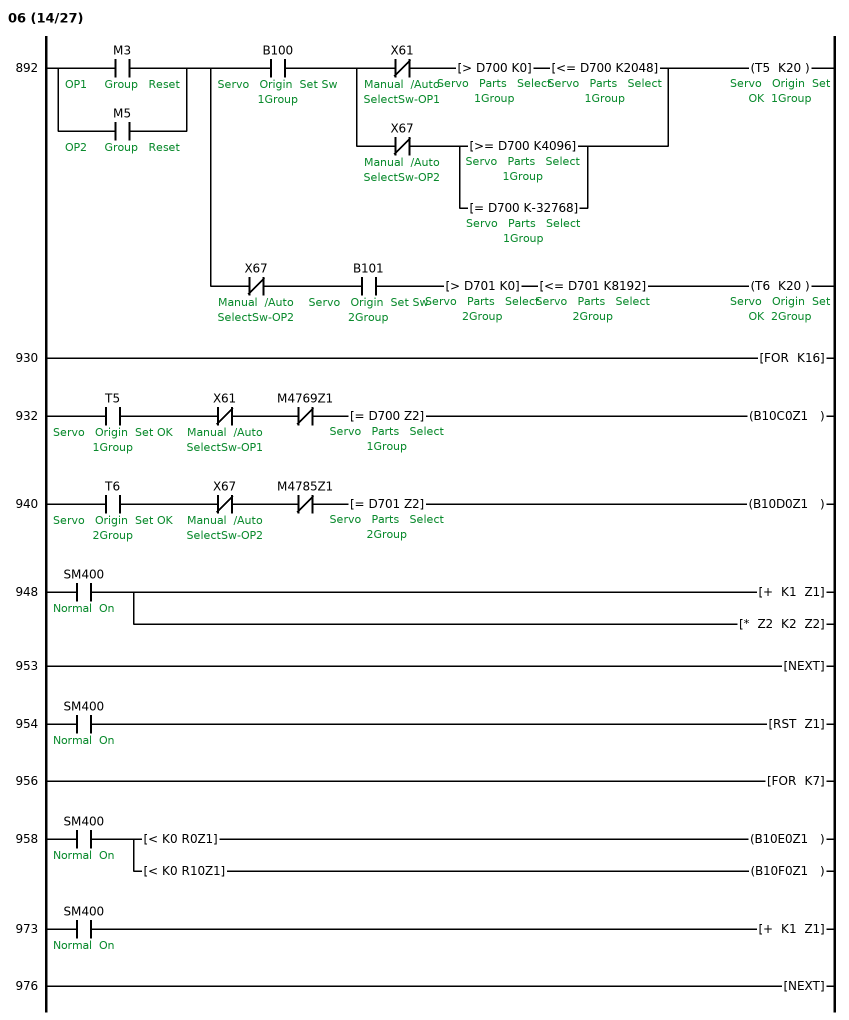
892   LD      M3  ; OP1     Group   Reset
      OR      M5  ; OP2     Group   Reset
      MPS
      AND     B100  ; Servo   Origin  Set Sw  1Group
      LDI     X61  ; Manual  /Auto   SelectSw-OP1
      AND>    D700 K0  ; Servo   Parts   Select  1Group
      AND<=   D700 K2048  ; Servo   Parts   Select  1Group
      LDI     X67  ; Manual  /Auto   SelectSw-OP2
      LD>=    D700 K4096  ; Servo   Parts   Select  1Group
      OR=     D700 K-32768  ; Servo   Parts   Select  1Group
      ANB
      ORB
      ANB
      OUT     T5 K20  ; Servo   Origin  Set OK  1Group
      MPP
      ANI     X67  ; Manual  /Auto   SelectSw-OP2
      AND     B101  ; Servo   Origin  Set Sw  2Group
      AND>    D701 K0  ; Servo   Parts   Select  2Group
      AND<=   D701 K8192  ; Servo   Parts   Select  2Group
      OUT     T6 K20  ; Servo   Origin  Set OK  2Group
930   FOR     K16
932   LD      T5  ; Servo   Origin  Set OK  1Group
      ANI     X61  ; Manual  /Auto   SelectSw-OP1
      ANI     M4769Z1
      AND=    D700 Z2  ; Servo   Parts   Select  1Group
      OUT     B10C0Z1
940   LD      T6  ; Servo   Origin  Set OK  2Group
      ANI     X67  ; Manual  /Auto   SelectSw-OP2
      ANI     M4785Z1
      AND=    D701 Z2  ; Servo   Parts   Select  2Group
      OUT     B10D0Z1
948   LD      SM400  ; Normal  On
      +       K1 Z1
      *       Z2 K2 Z2
953   NEXT
954   LD      SM400  ; Normal  On
      RST     Z1
956   FOR     K7
958   LD      SM400  ; Normal  On
      MPS
      AND<    K0 R0Z1
      OUT     B10E0Z1
      MPP
      AND<    K0 R10Z1
      OUT     B10F0Z1
973   LD      SM400  ; Normal  On
      +       K1 Z1
976   NEXT
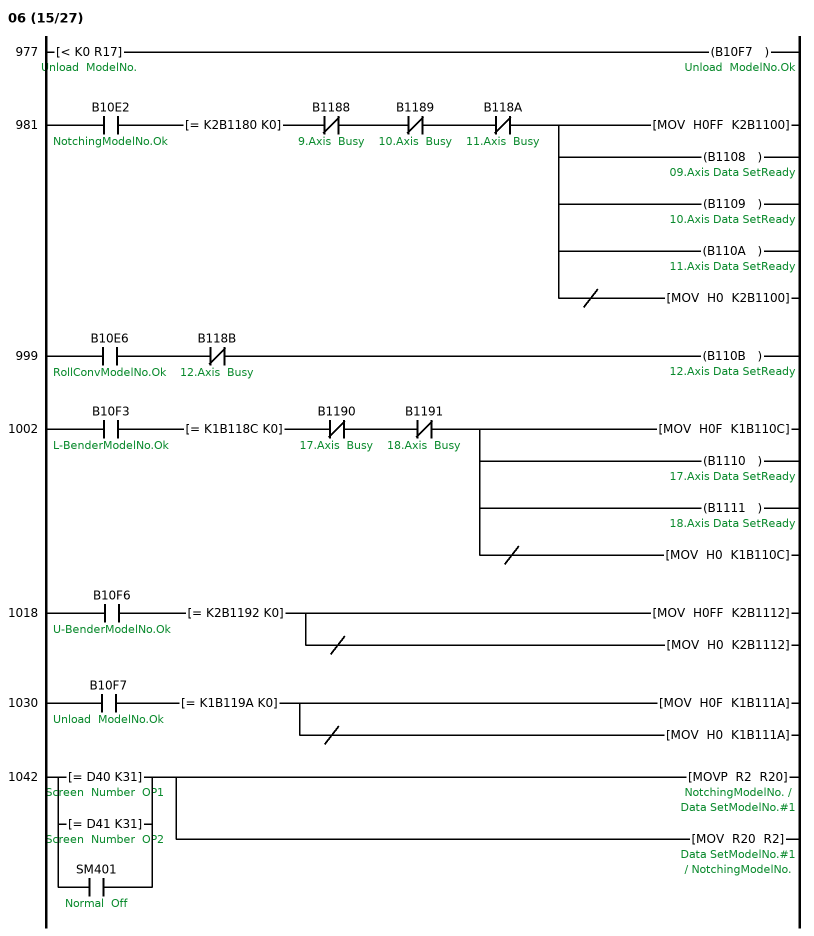
977   LD<     K0 R17  ; Unload  ModelNo.
      OUT     B10F7  ; Unload  ModelNo.Ok
981   LD      B10E2  ; NotchingModelNo.Ok
      AND=    K2B1180 K0  ; 1.Axis  Busy
      ANI     B1188  ; 9.Axis  Busy
      ANI     B1189  ; 10.Axis  Busy
      ANI     B118A  ; 11.Axis  Busy
      MOV     H0FF K2B1100  ; 01.Axis Data SetReady
      OUT     B1108  ; 09.Axis Data SetReady
      OUT     B1109  ; 10.Axis Data SetReady
      OUT     B110A  ; 11.Axis Data SetReady
      INV
      MOV     H0 K2B1100
999   LD      B10E6  ; RollConvModelNo.Ok
      ANI     B118B  ; 12.Axis  Busy
      OUT     B110B  ; 12.Axis Data SetReady
1002  LD      B10F3  ; L-BenderModelNo.Ok
      AND=    K1B118C K0  ; 13.Axis  Busy
      ANI     B1190  ; 17.Axis  Busy
      ANI     B1191  ; 18.Axis  Busy
      MOV     H0F K1B110C  ; 13.Axis Data SetReady
      OUT     B1110  ; 17.Axis Data SetReady
      OUT     B1111  ; 18.Axis Data SetReady
      INV
      MOV     H0 K1B110C
1018  LD      B10F6  ; U-BenderModelNo.Ok
      AND=    K2B1192 K0  ; 19.Axis  Busy
      MOV     H0FF K2B1112  ; 19.Axis Data SetReady
      INV
      MOV     H0 K2B1112
1030  LD      B10F7  ; Unload  ModelNo.Ok
      AND=    K1B119A K0  ; 27.Axis  Busy
      MOV     H0F K1B111A  ; 27.Axis Data SetReady
      INV
      MOV     H0 K1B111A
1042  LD=     D40 K31  ; Screen  Number  OP1
      OR=     D41 K31  ; Screen  Number  OP2
      OR      SM401  ; Normal  Off
      MOVP    R2 R20  ; NotchingModelNo. / Data SetModelNo.#1
      MOV     R20 R2
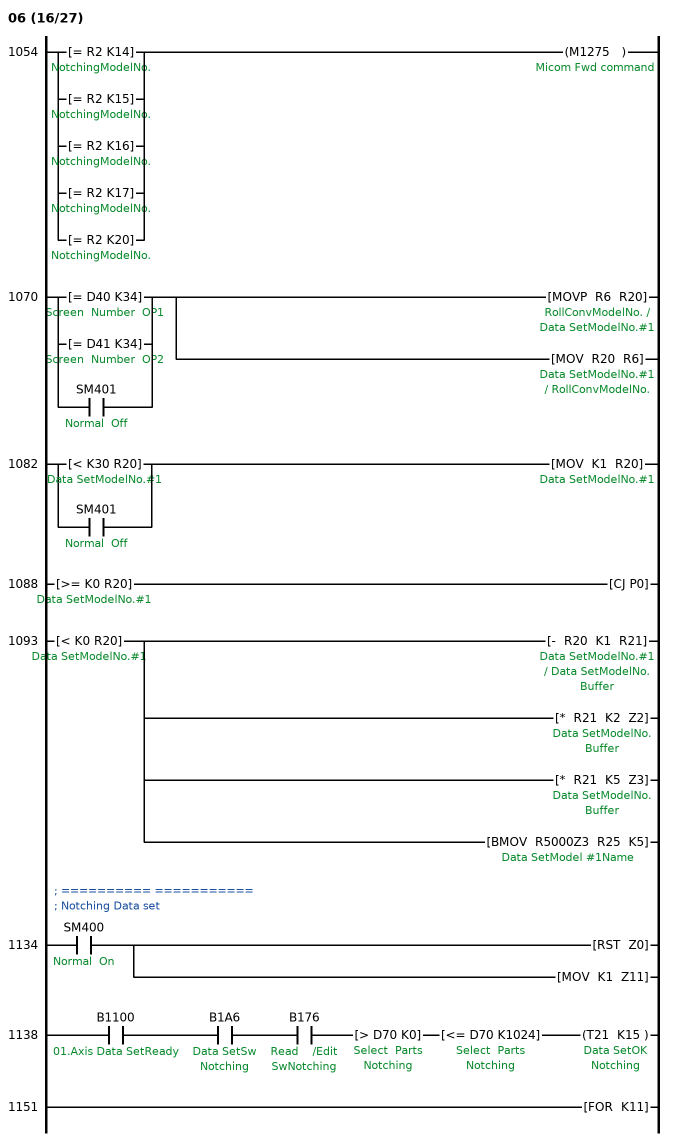
1054  LD=     R2 K14  ; NotchingModelNo.
      OR=     R2 K15  ; NotchingModelNo.
      OR=     R2 K16  ; NotchingModelNo.
      OR=     R2 K17  ; NotchingModelNo.
      OR=     R2 K20  ; NotchingModelNo.
      OUT     M1275  ; Micom Fwd command
1070  LD=     D40 K34  ; Screen  Number  OP1
      OR=     D41 K34  ; Screen  Number  OP2
      OR      SM401  ; Normal  Off
      MOVP    R6 R20  ; RollConvModelNo.
      MOV     R20 R6
1082  LD<     K30 R20  ; Data SetModelNo.#1
      OR      SM401  ; Normal  Off
      MOV     K1 R20
1088  LD>=    K0 R20  ; Data SetModelNo.#1
      CJ      P0  ; Jump
1093  LD<     K0 R20  ; Data SetModelNo.#1
      -       R20 K1 R21  ; Data SetModelNo.Buffer
      *       R21 K2 Z2
      *       R21 K5 Z3
      BMOV    R5000Z3 R25 K5  ; Data SetModel #1Name
; ========== ===========
; Notching Data set
1134  LD      SM400  ; Normal  On
      RST     Z0
      MOV     K1 Z11
1138  LD      B1100  ; 01.Axis Data SetReady
      AND     B1A6  ; Data SetSw      Notching
      AND     B176  ; Read    /Edit SwNotching
      AND>    D70 K0  ; Select  Parts   Notching
      AND<=   D70 K1024  ; Select  Parts   Notching
      OUT     T21 K15  ; Data SetOK      Notching
1151  FOR     K11
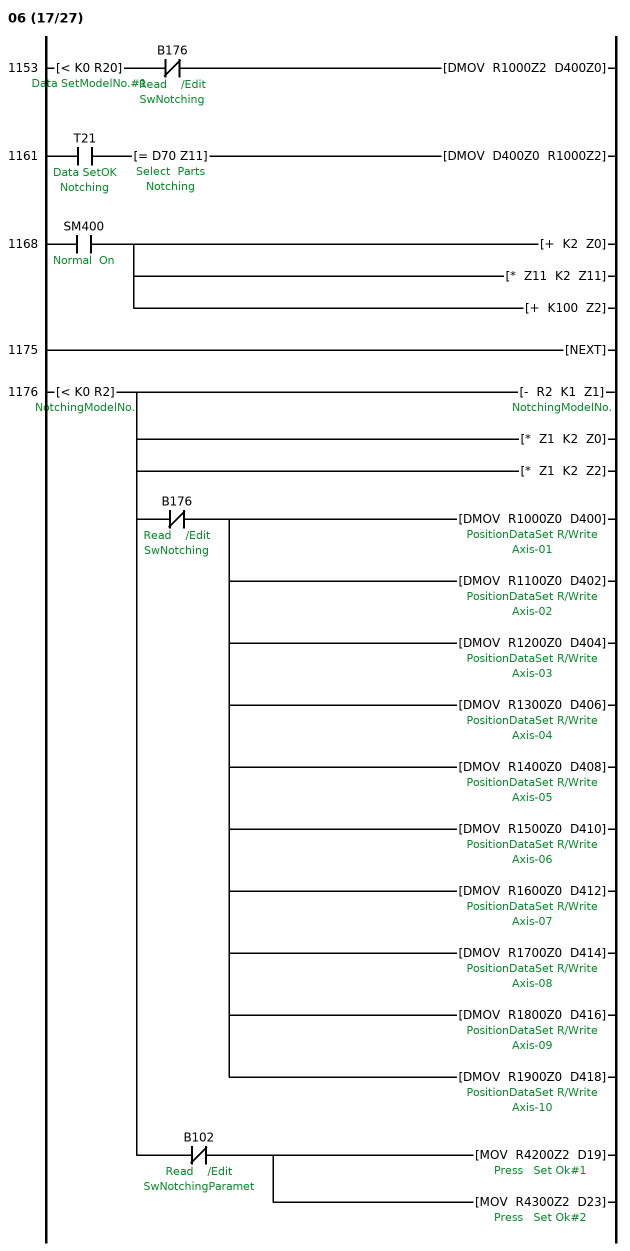
1153  LD<     K0 R20  ; Data SetModelNo.#1
      ANI     B176  ; Read    /Edit SwNotching
      DMOV    R1000Z2 D400Z0
1161  LD      T21  ; Data SetOK      Notching
      AND=    D70 Z11  ; Select  Parts   Notching
      DMOV    D400Z0 R1000Z2
1168  LD      SM400  ; Normal  On
      +       K2 Z0
      *       Z11 K2 Z11
      +       K100 Z2
1175  NEXT
1176  LD<     K0 R2  ; NotchingModelNo.
      -       R2 K1 Z1
      *       Z1 K2 Z0
      *       Z1 K2 Z2
      MPS
      ANI     B176  ; Read    /Edit SwNotching
      DMOV    R1000Z0 D400  ; PositionDataSet R/Write Axis-01
      DMOV    R1100Z0 D402  ; PositionDataSet R/Write Axis-02
      DMOV    R1200Z0 D404  ; PositionDataSet R/Write Axis-03
      DMOV    R1300Z0 D406  ; PositionDataSet R/Write Axis-04
      DMOV    R1400Z0 D408  ; PositionDataSet R/Write Axis-05
      DMOV    R1500Z0 D410  ; PositionDataSet R/Write Axis-06
      DMOV    R1600Z0 D412  ; PositionDataSet R/Write Axis-07
      DMOV    R1700Z0 D414  ; PositionDataSet R/Write Axis-08
      DMOV    R1800Z0 D416  ; PositionDataSet R/Write Axis-09
      DMOV    R1900Z0 D418  ; PositionDataSet R/Write Axis-10
      MPP
      ANI     B102  ; Read    /Edit SwNotchingParamet
      MOV     R4200Z2 D19  ; Press   Set Ok#1
      MOV     R4300Z2 D23  ; Press   Set Ok#2
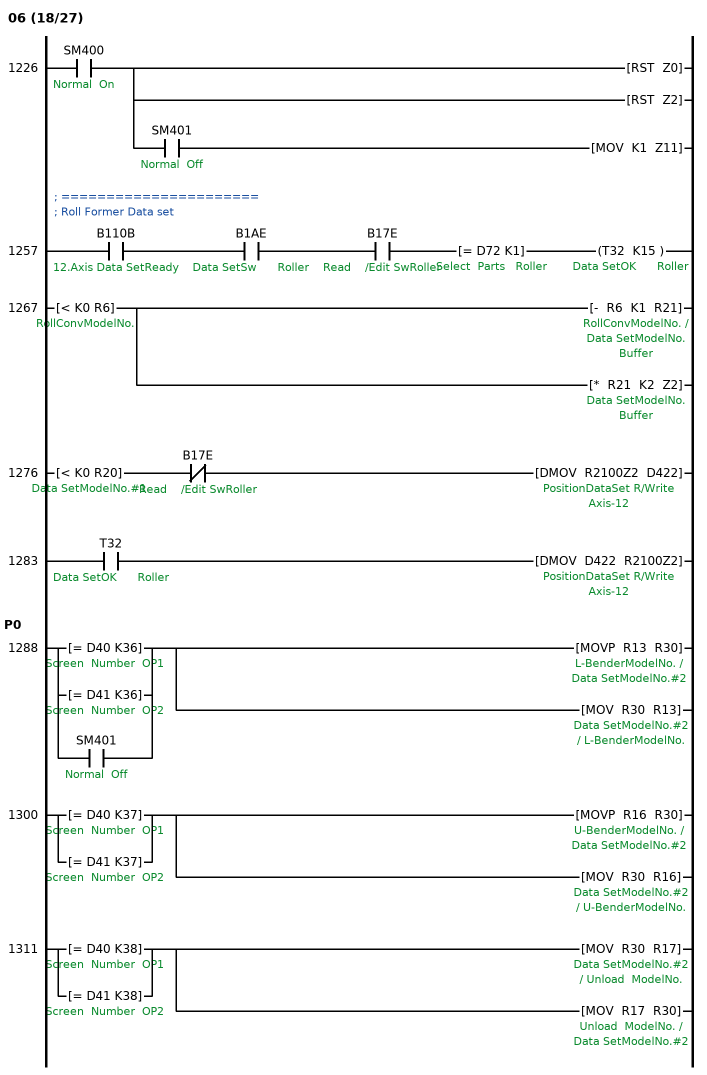
1226  LD      SM400  ; Normal  On
      RST     Z0
      RST     Z2
      AND     SM401  ; Normal  Off
      MOV     K1 Z11
; ======================
; Roll Former Data set
1257  LD      B110B  ; 12.Axis Data SetReady
      AND     B1AE  ; Data SetSw      Roller
      AND     B17E  ; Read    /Edit SwRoller
      AND=    D72 K1  ; Select  Parts   Roller
      OUT     T32 K15  ; Data SetOK      Roller
1267  LD<     K0 R6  ; RollConvModelNo.
      -       R6 K1 R21
      *       R21 K2 Z2
1276  LD<     K0 R20  ; Data SetModelNo.#1
      ANI     B17E  ; Read    /Edit SwRoller
      DMOV    R2100Z2 D422  ; PositionDataSet R/Write Axis-12
1283  LD      T32  ; Data SetOK      Roller
      DMOV    D422 R2100Z2
      P0
1288  LD=     D40 K36  ; Screen  Number  OP1
      OR=     D41 K36  ; Screen  Number  OP2
      OR      SM401  ; Normal  Off
      MOVP    R13 R30  ; L-BenderModelNo. / Data SetModelNo.#2
      MOV     R30 R13
1300  LD=     D40 K37  ; Screen  Number  OP1
      OR=     D41 K37  ; Screen  Number  OP2
      MOVP    R16 R30  ; U-BenderModelNo.
      MOV     R30 R16
1311  LD=     D40 K38  ; Screen  Number  OP1
      OR=     D41 K38  ; Screen  Number  OP2
      MOV     R30 R17
      MOV     R17 R30
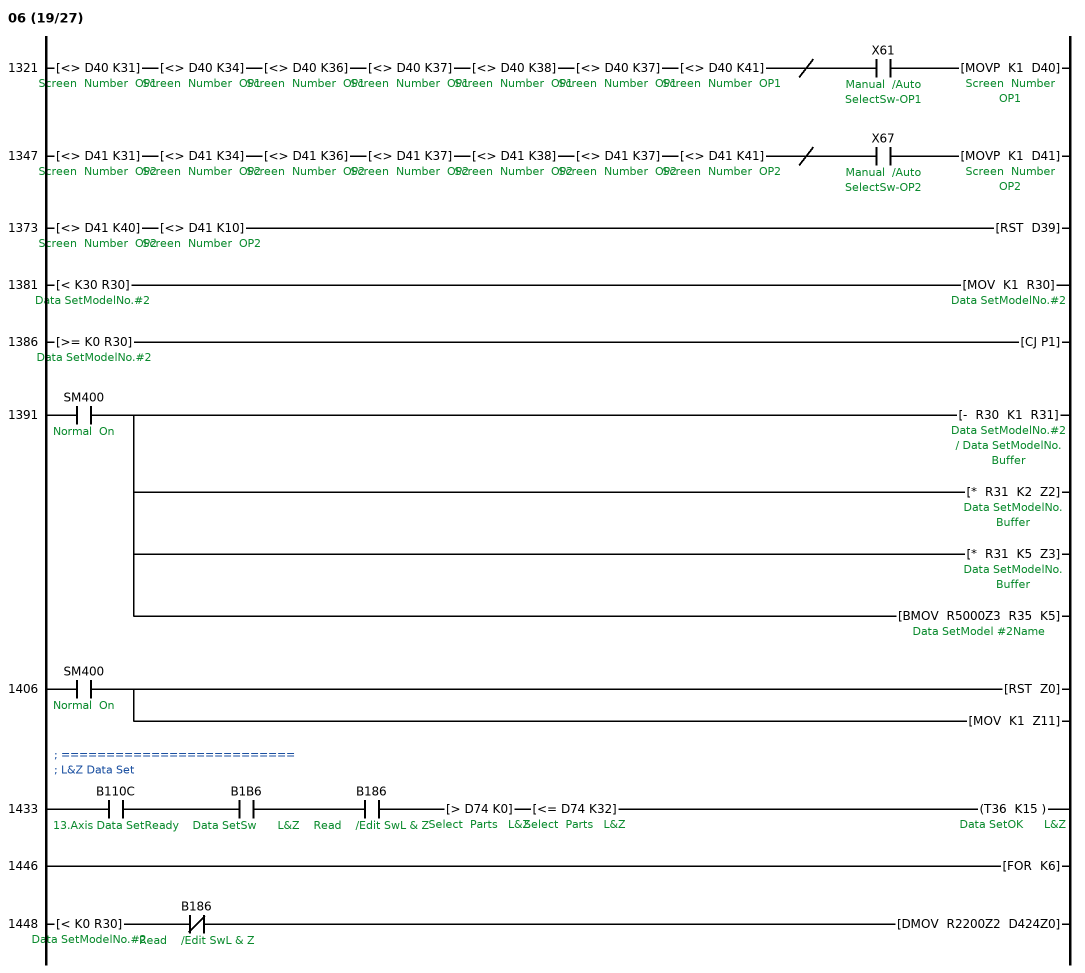
1321  LD<>    D40 K31  ; Screen  Number  OP1
      AND<>   D40 K34  ; Screen  Number  OP1
      AND<>   D40 K36  ; Screen  Number  OP1
      AND<>   D40 K37  ; Screen  Number  OP1
      AND<>   D40 K38  ; Screen  Number  OP1
      AND<>   D40 K37  ; Screen  Number  OP1
      AND<>   D40 K41  ; Screen  Number  OP1
      INV
      AND     X61  ; Manual  /Auto   SelectSw-OP1
      MOVP    K1 D40
1347  LD<>    D41 K31  ; Screen  Number  OP2
      AND<>   D41 K34  ; Screen  Number  OP2
      AND<>   D41 K36  ; Screen  Number  OP2
      AND<>   D41 K37  ; Screen  Number  OP2
      AND<>   D41 K38  ; Screen  Number  OP2
      AND<>   D41 K37  ; Screen  Number  OP2
      AND<>   D41 K41  ; Screen  Number  OP2
      INV
      AND     X67  ; Manual  /Auto   SelectSw-OP2
      MOVP    K1 D41
1373  LD<>    D41 K40  ; Screen  Number  OP2
      AND<>   D41 K10  ; Screen  Number  OP2
      RST     D39
1381  LD<     K30 R30  ; Data SetModelNo.#2
      MOV     K1 R30
1386  LD>=    K0 R30  ; Data SetModelNo.#2
      CJ      P1  ; Jump
1391  LD      SM400  ; Normal  On
      -       R30 K1 R31  ; Data SetModelNo.Buffer
      *       R31 K2 Z2
      *       R31 K5 Z3
      BMOV    R5000Z3 R35 K5  ; Data SetModel #2Name
1406  LD      SM400  ; Normal  On
      RST     Z0
      MOV     K1 Z11
; ==========================
; L&Z Data Set
1433  LD      B110C  ; 13.Axis Data SetReady
      AND     B1B6  ; Data SetSw      L&Z
      AND     B186  ; Read    /Edit SwL & Z
      AND>    D74 K0  ; Select  Parts   L&Z
      AND<=   D74 K32  ; Select  Parts   L&Z
      OUT     T36 K15  ; Data SetOK      L&Z
1446  FOR     K6
1448  LD<     K0 R30  ; Data SetModelNo.#2
      ANI     B186  ; Read    /Edit SwL & Z
      DMOV    R2200Z2 D424Z0
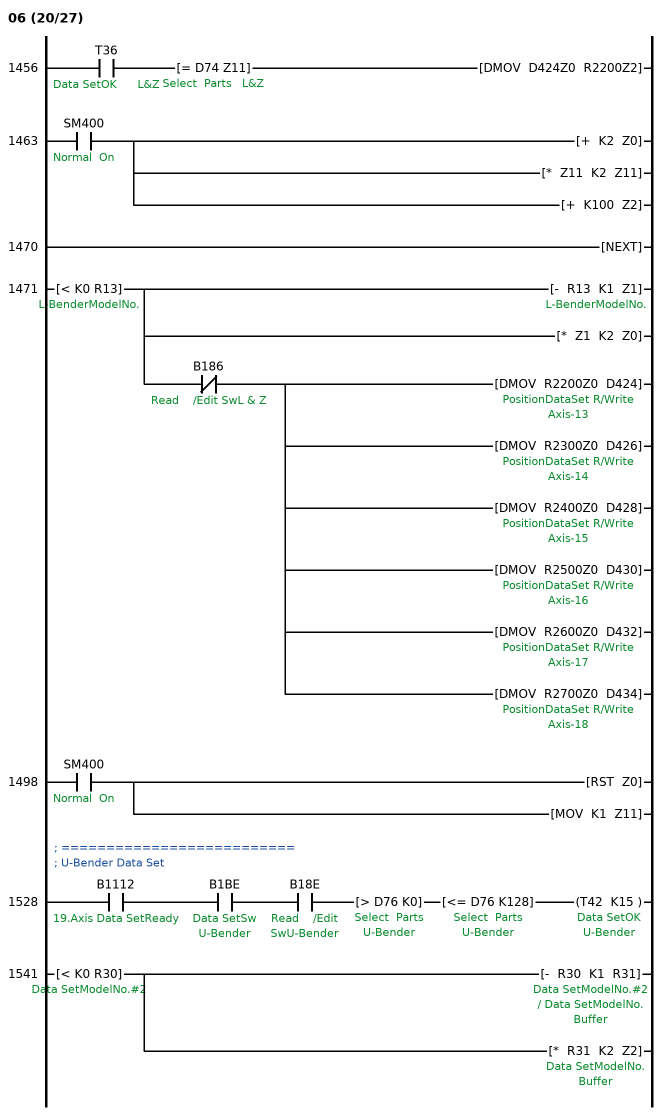
1456  LD      T36  ; Data SetOK      L&Z
      AND=    D74 Z11  ; Select  Parts   L&Z
      DMOV    D424Z0 R2200Z2
1463  LD      SM400  ; Normal  On
      +       K2 Z0
      *       Z11 K2 Z11
      +       K100 Z2
1470  NEXT
1471  LD<     K0 R13  ; L-BenderModelNo.
      -       R13 K1 Z1
      *       Z1 K2 Z0
      ANI     B186  ; Read    /Edit SwL & Z
      DMOV    R2200Z0 D424  ; PositionDataSet R/Write Axis-13
      DMOV    R2300Z0 D426  ; PositionDataSet R/Write Axis-14
      DMOV    R2400Z0 D428  ; PositionDataSet R/Write Axis-15
      DMOV    R2500Z0 D430  ; PositionDataSet R/Write Axis-16
      DMOV    R2600Z0 D432  ; PositionDataSet R/Write Axis-17
      DMOV    R2700Z0 D434  ; PositionDataSet R/Write Axis-18
1498  LD      SM400  ; Normal  On
      RST     Z0
      MOV     K1 Z11
; ==========================
; U-Bender Data Set
1528  LD      B1112  ; 19.Axis Data SetReady
      AND     B1BE  ; Data SetSw      U-Bender
      AND     B18E  ; Read    /Edit SwU-Bender
      AND>    D76 K0  ; Select  Parts   U-Bender
      AND<=   D76 K128  ; Select  Parts   U-Bender
      OUT     T42 K15  ; Data SetOK      U-Bender
1541  LD<     K0 R30  ; Data SetModelNo.#2
      -       R30 K1 R31
      *       R31 K2 Z2
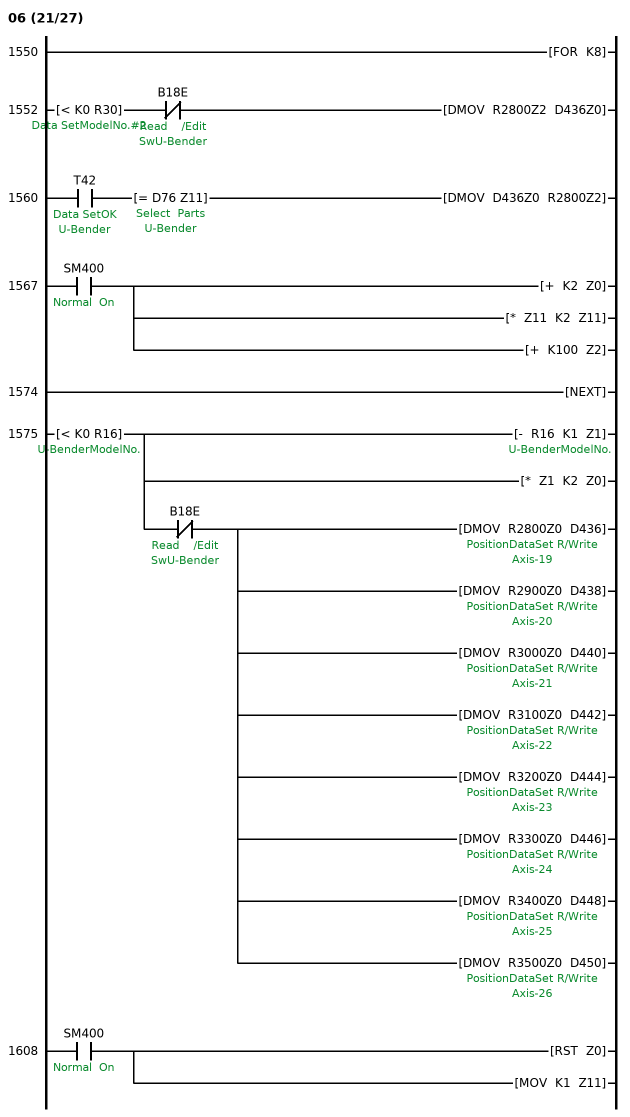
1550  FOR     K8
1552  LD<     K0 R30  ; Data SetModelNo.#2
      ANI     B18E  ; Read    /Edit SwU-Bender
      DMOV    R2800Z2 D436Z0
1560  LD      T42  ; Data SetOK      U-Bender
      AND=    D76 Z11  ; Select  Parts   U-Bender
      DMOV    D436Z0 R2800Z2
1567  LD      SM400  ; Normal  On
      +       K2 Z0
      *       Z11 K2 Z11
      +       K100 Z2
1574  NEXT
1575  LD<     K0 R16  ; U-BenderModelNo.
      -       R16 K1 Z1
      *       Z1 K2 Z0
      ANI     B18E  ; Read    /Edit SwU-Bender
      DMOV    R2800Z0 D436  ; PositionDataSet R/Write Axis-19
      DMOV    R2900Z0 D438  ; PositionDataSet R/Write Axis-20
      DMOV    R3000Z0 D440  ; PositionDataSet R/Write Axis-21
      DMOV    R3100Z0 D442  ; PositionDataSet R/Write Axis-22
      DMOV    R3200Z0 D444  ; PositionDataSet R/Write Axis-23
      DMOV    R3300Z0 D446  ; PositionDataSet R/Write Axis-24
      DMOV    R3400Z0 D448  ; PositionDataSet R/Write Axis-25
      DMOV    R3500Z0 D450  ; PositionDataSet R/Write Axis-26
1608  LD      SM400  ; Normal  On
      RST     Z0
      MOV     K1 Z11
